C01840=1183.725,109.881,-51.815,-178.781,6.157,148.748
C01841=1183.720,110.129,-51.834,-178.778,6.158,148.748
C01842=1183.715,110.379,-51.854,-178.775,6.159,148.747
C01843=1183.710,110.628,-51.872,-178.773,6.160,148.747
C01844=1183.706,110.878,-51.891,-178.770,6.162,148.746
C01845=1183.701,111.126,-51.910,-178.767,6.163,148.746
C01846=1183.696,111.376,-51.929,-178.765,6.164,148.745
C01847=1183.691,111.625,-51.948,-178.762,6.166,148.745
C01848=1183.687,111.874,-51.967,-178.760,6.167,148.744
C01849=1183.682,112.123,-51.986,-178.757,6.168,148.744
C01850=1183.677,112.373,-52.005,-178.754,6.170,148.743
C01851=1183.672,112.622,-52.024,-178.752,6.171,148.743
C01852=1183.668,112.871,-52.043,-178.749,6.172,148.742
C01853=1183.662,113.120,-52.063,-178.746,6.174,148.742
C01854=1183.658,113.370,-52.081,-178.744,6.175,148.741
C01855=1183.653,113.619,-52.100,-178.741,6.177,148.741
C01856=1183.648,113.869,-52.120,-178.738,6.177,148.740
C01857=1183.643,114.117,-52.139,-178.736,6.179,148.740
C01858=1183.639,114.367,-52.158,-178.733,6.181,148.740
C01859=1183.634,114.616,-52.176,-178.730,6.181,148.739
C01860=1183.629,114.865,-52.196,-178.728,6.183,148.739
C01861=1183.624,115.114,-52.215,-178.726,6.184,148.738
C01862=1183.619,115.363,-52.234,-178.722,6.185,148.737
C01863=1183.614,115.612,-52.254,-178.720,6.187,148.737
C01864=1183.609,115.862,-52.273,-178.718,6.188,148.737
C01865=1183.605,116.110,-52.292,-178.714,6.189,148.736
C01866=1183.600,116.361,-52.311,-178.712,6.191,148.736
C01867=1183.594,116.610,-52.330,-178.710,6.192,148.735
C01868=1183.590,116.859,-52.349,-178.706,6.193,148.735
C01869=1183.585,117.108,-52.368,-178.704,6.195,148.734
C01870=1183.580,117.357,-52.388,-178.701,6.196,148.734
C01871=1183.576,117.607,-52.408,-178.698,6.197,148.733
C01872=1183.571,117.855,-52.427,-178.696,6.198,148.733
C01873=1183.566,118.105,-52.446,-178.693,6.200,148.732
C01874=1183.561,118.354,-52.465,-178.690,6.201,148.732
C01875=1183.556,118.603,-52.485,-178.688,6.202,148.731
C01876=1183.552,118.852,-52.504,-178.685,6.204,148.731
C01877=1183.547,119.101,-52.523,-178.683,6.206,148.731
C01878=1183.542,119.351,-52.543,-178.680,6.206,148.730
C01879=1183.537,119.600,-52.562,-178.677,6.208,148.729
C01880=1183.533,119.849,-52.581,-178.675,6.210,148.729
C01881=1183.527,120.098,-52.601,-178.672,6.210,148.728
C01882=1183.523,120.348,-52.620,-178.669,6.212,148.728
C01883=1183.518,120.597,-52.640,-178.667,6.214,148.728
C01884=1183.513,120.846,-52.659,-178.664,6.215,148.727
C01885=1183.509,121.095,-52.679,-178.661,6.216,148.727
C01886=1183.504,121.344,-52.699,-178.659,6.218,148.726
C01887=1183.499,121.593,-52.718,-178.657,6.219,148.726
C01888=1183.494,121.843,-52.738,-178.653,6.220,148.725
C01889=1183.489,122.092,-52.757,-178.651,6.222,148.725
C01890=1183.484,122.341,-52.777,-178.649,6.223,148.724
C01891=1183.480,122.590,-52.796,-178.645,6.224,148.724
C01892=1183.475,122.840,-52.815,-178.643,6.226,148.723
C01893=1183.470,123.088,-52.835,-178.641,6.227,148.723
C01894=1183.465,123.338,-52.855,-178.637,6.228,148.722
C01895=1183.461,123.587,-52.875,-178.635,6.230,148.722
C01896=1183.455,123.836,-52.894,-178.633,6.231,148.722
C01897=1183.451,124.086,-52.914,-178.630,6.233,148.721
C01898=1183.446,124.335,-52.934,-178.627,6.234,148.721
C01899=1183.441,124.584,-52.953,-178.624,6.236,148.720
C01900=1183.437,124.833,-52.972,-178.622,6.237,148.720
C01901=1183.432,125.082,-52.992,-178.619,6.239,148.719
C01902=1183.427,125.331,-53.012,-178.616,6.240,148.719
C01903=1183.422,125.580,-53.032,-178.614,6.241,148.718
C01904=1183.417,125.830,-53.051,-178.611,6.243,148.718
C01905=1183.413,126.079,-53.072,-178.608,6.244,148.717
C01906=1183.408,126.328,-53.091,-178.606,6.245,148.717
C01907=1183.403,126.577,-53.111,-178.603,6.247,148.716
C01908=1183.399,126.826,-53.131,-178.600,6.249,148.716
C01909=1183.394,127.076,-53.151,-178.597,6.250,148.715
C01910=1183.388,127.325,-53.170,-178.595,6.251,148.715
C01911=1183.384,127.574,-53.190,-178.592,6.253,148.715
C01912=1183.379,127.823,-53.210,-178.590,6.254,148.714
C01913=1183.375,128.073,-53.230,-178.587,6.255,148.714
C01914=1183.369,128.321,-53.250,-178.584,6.257,148.713
C01915=1183.365,128.570,-53.269,-178.582,6.258,148.713
C01916=1183.360,128.819,-53.290,-178.579,6.260,148.712
C01917=1183.356,129.069,-53.309,-178.576,6.261,148.712
C01918=1183.350,129.318,-53.329,-178.574,6.263,148.711
C01919=1183.346,129.567,-53.349,-178.571,6.264,148.711
C01920=1183.341,129.816,-53.369,-178.569,6.265,148.711
C01921=1183.337,130.065,-53.389,-178.566,6.267,148.710
C01922=1183.332,130.315,-53.409,-178.563,6.268,148.710
C01923=1183.327,130.563,-53.429,-178.560,6.270,148.709
C01924=1183.321,130.813,-53.449,-178.558,6.271,148.709
C01925=1183.317,131.062,-53.469,-178.555,6.272,148.708
C01926=1183.312,131.312,-53.489,-178.552,6.274,148.708
C01927=1183.308,131.560,-53.509,-178.550,6.276,148.707
C01928=1183.302,131.809,-53.529,-178.548,6.277,148.707
C01929=1183.298,132.058,-53.549,-178.544,6.278,148.706
C01930=1183.292,132.327,-53.571,-178.542,6.280,148.706
C01931=1183.288,132.595,-53.593,-178.539,6.282,148.706
C01932=1183.282,132.864,-53.614,-178.536,6.283,148.705
C01933=1183.277,133.133,-53.635,-178.533,6.285,148.705
C01934=1183.273,133.382,-53.656,-178.530,6.287,148.704
C01935=1183.268,133.631,-53.676,-178.528,6.287,148.704
C01936=1183.263,133.881,-53.696,-178.525,6.289,148.703
C01937=1183.258,134.130,-53.717,-178.522,6.291,148.703
C01938=1183.254,134.379,-53.736,-178.520,6.293,148.702
C01939=1183.249,134.628,-53.757,-178.517,6.293,148.702
C01940=1183.244,134.876,-53.777,-178.514,6.295,148.701
C01941=1183.239,135.126,-53.797,-178.512,6.297,148.701
C01942=1183.234,135.375,-53.817,-178.509,6.298,148.701
C01943=1183.230,135.624,-53.838,-178.507,6.299,148.700
C01944=1183.225,135.873,-53.858,-178.504,6.301,148.700
C01945=1183.220,136.123,-53.878,-178.501,6.302,148.699
C01946=1183.215,136.372,-53.899,-178.498,6.304,148.699
C01947=1183.211,136.621,-53.919,-178.496,6.306,148.698
C01948=1183.206,136.870,-53.939,-178.493,6.307,148.698
C01949=1183.201,137.120,-53.960,-178.490,6.308,148.697
C01950=1183.197,137.369,-53.980,-178.488,6.310,148.697
C01951=1183.192,137.617,-54.000,-178.485,6.312,148.697
C01952=1183.187,137.866,-54.020,-178.483,6.313,148.696
C01953=1183.182,138.116,-54.041,-178.480,6.315,148.696
C01954=1183.177,138.365,-54.061,-178.477,6.316,148.695
C01955=1183.173,138.614,-54.081,-178.474,6.318,148.695
C01956=1183.168,138.863,-54.102,-178.472,6.319,148.695
C01957=1183.163,139.112,-54.123,-178.469,6.320,148.694
C01958=1183.159,139.361,-54.143,-178.467,6.322,148.694
C01959=1183.153,139.611,-54.163,-178.464,6.324,148.693
C01960=1183.149,139.860,-54.184,-178.461,6.325,148.693
C01961=1183.144,140.109,-54.204,-178.459,6.326,148.692
C01962=1183.139,140.358,-54.225,-178.456,6.328,148.692
C01963=1183.135,140.607,-54.245,-178.453,6.330,148.692
C01964=1183.130,140.856,-54.266,-178.451,6.332,148.691
C01965=1183.125,141.105,-54.287,-178.447,6.333,148.691
C01966=1183.121,141.354,-54.307,-178.445,6.334,148.690
C01967=1183.116,141.603,-54.328,-178.443,6.336,148.690
C01968=1183.111,141.852,-54.349,-178.440,6.337,148.689
C01969=1183.107,142.101,-54.369,-178.437,6.339,148.689
C01970=1183.101,142.350,-54.390,-178.434,6.341,148.688
C01971=1183.097,142.599,-54.410,-178.431,6.342,148.688
C01972=1183.092,142.849,-54.431,-178.429,6.343,148.688
C01973=1183.087,143.098,-54.452,-178.427,6.345,148.687
C01974=1183.083,143.346,-54.472,-178.424,6.347,148.687
C01975=1183.078,143.596,-54.493,-178.421,6.349,148.686
C01976=1183.073,143.845,-54.513,-178.418,6.350,148.686
C01977=1183.068,144.094,-54.534,-178.416,6.351,148.685
C01978=1183.064,144.343,-54.555,-178.413,6.353,148.685
C01979=1183.059,144.592,-54.576,-178.411,6.354,148.685
C01980=1183.055,144.842,-54.596,-178.408,6.356,148.684
C01981=1183.050,145.091,-54.617,-178.405,6.358,148.684
C01982=1183.045,145.340,-54.638,-178.402,6.360,148.684
C01983=1183.040,145.589,-54.659,-178.400,6.360,148.683
C01984=1183.036,145.838,-54.679,-178.397,6.362,148.683
C01985=1183.031,146.087,-54.701,-178.395,6.364,148.682
C01986=1183.026,146.336,-54.721,-178.392,6.366,148.682
C01987=1183.021,146.585,-54.742,-178.389,6.367,148.681
C01988=1183.017,146.834,-54.762,-178.386,6.369,148.681
C01989=1183.011,147.083,-54.783,-178.384,6.370,148.681
C01990=1183.006,147.333,-54.804,-178.381,6.371,148.680
C01991=1183.003,147.582,-54.826,-178.378,6.373,148.680
C01992=1182.998,147.831,-54.847,-178.376,6.375,148.679
C01993=1182.993,148.080,-54.867,-178.373,6.377,148.679
C01994=1182.988,148.329,-54.888,-178.370,6.378,148.678
C01995=1182.984,148.577,-54.909,-178.368,6.380,148.678
C01996=1182.979,148.827,-54.930,-178.366,6.381,148.678
C01997=1182.973,149.076,-54.951,-178.362,6.383,148.677
C01998=1182.970,149.326,-54.972,-178.360,6.384,148.677
C01999=1182.965,149.574,-54.994,-178.357,6.386,148.676
C02000=1182.960,149.823,-55.014,-178.354,6.388,148.676
C02001=1182.955,150.072,-55.035,-178.352,6.390,148.676
C02002=1182.950,150.321,-55.057,-178.349,6.391,148.675
C02003=1182.945,150.570,-55.078,-178.347,6.392,148.675
C02004=1182.941,150.819,-55.098,-178.344,6.394,148.674
C02005=1182.936,151.069,-55.120,-178.342,6.396,148.674
C02006=1182.931,151.318,-55.141,-178.338,6.397,148.673
C02007=1182.927,151.567,-55.161,-178.336,6.399,148.673
C02008=1182.922,151.815,-55.183,-178.333,6.401,148.673
C02009=1182.917,152.065,-55.204,-178.330,6.403,148.672
C02010=1182.913,152.314,-55.225,-178.328,6.404,148.672
C02011=1182.908,152.563,-55.246,-178.325,6.405,148.672
C02012=1182.903,152.812,-55.267,-178.323,6.407,148.671
C02013=1182.898,153.061,-55.289,-178.320,6.409,148.671
C02014=1182.894,153.310,-55.309,-178.317,6.411,148.670
C02015=1182.889,153.559,-55.331,-178.314,6.412,148.670
C02016=1182.884,153.808,-55.352,-178.312,6.414,148.669
C02017=1182.879,154.057,-55.374,-178.309,6.416,148.669
C02018=1182.875,154.306,-55.394,-178.306,6.417,148.669
C02019=1182.871,154.555,-55.416,-178.304,6.418,148.668
C02020=1182.865,154.805,-55.437,-178.301,6.420,148.668
C02021=1182.861,155.053,-55.459,-178.299,6.422,148.668
C02022=1182.856,155.302,-55.480,-178.296,6.424,148.667
C02023=1182.852,155.552,-55.502,-178.293,6.425,148.667
C02024=1182.847,155.801,-55.523,-178.291,6.427,148.666
C02025=1182.842,156.049,-55.544,-178.288,6.429,148.666
C02026=1182.837,156.299,-55.565,-178.285,6.431,148.666
C02027=1182.832,156.548,-55.587,-178.282,6.432,148.665
C02028=1182.828,156.796,-55.608,-178.279,6.434,148.665
C02029=1182.823,157.046,-55.629,-178.277,6.436,148.664
C02030=1182.819,157.295,-55.651,-178.275,6.437,148.664
C02031=1182.814,157.544,-55.672,-178.272,6.438,148.664
C02032=1182.809,157.793,-55.694,-178.269,6.440,148.663
C02033=1182.804,158.041,-55.716,-178.267,6.442,148.663
C02034=1182.799,158.311,-55.738,-178.264,6.444,148.662
C02035=1182.794,158.580,-55.762,-178.261,6.445,148.662
C02036=1182.789,158.848,-55.785,-178.257,6.448,148.661
C02037=1182.784,159.118,-55.809,-178.255,6.449,148.661
C02038=1182.779,159.367,-55.831,-178.252,6.451,148.661
C02039=1182.774,159.616,-55.852,-178.249,6.453,148.660
C02040=1182.770,159.865,-55.873,-178.247,6.455,148.660
C02041=1182.766,160.114,-55.895,-178.244,6.456,148.660
C02042=1182.761,160.363,-55.916,-178.242,6.457,148.659
C02043=1182.756,160.612,-55.937,-178.239,6.459,148.659
C02044=1182.752,160.861,-55.959,-178.237,6.461,148.658
C02045=1182.747,161.110,-55.981,-178.234,6.463,148.658
C02046=1182.742,161.358,-56.003,-178.231,6.464,148.658
C02047=1182.738,161.608,-56.025,-178.229,6.466,148.657
C02048=1182.732,161.857,-56.046,-178.226,6.468,148.657
C02049=1182.728,162.106,-56.068,-178.223,6.470,148.657
C02050=1182.723,162.355,-56.090,-178.220,6.471,148.656
C02051=1182.718,162.604,-56.111,-178.217,6.473,148.656
C02052=1182.714,162.853,-56.133,-178.215,6.475,148.655
C02053=1182.709,163.102,-56.155,-178.212,6.477,148.655
C02054=1182.705,163.352,-56.176,-178.209,6.478,148.655
C02055=1182.700,163.600,-56.198,-178.207,6.480,148.654
C02056=1182.695,163.849,-56.220,-178.204,6.482,148.654
C02057=1182.691,164.098,-56.242,-178.201,6.484,148.653
C02058=1182.686,164.347,-56.263,-178.199,6.485,148.653
C02059=1182.681,164.596,-56.285,-178.196,6.487,148.653
C02060=1182.676,164.845,-56.308,-178.193,6.489,148.652
C02061=1182.672,165.095,-56.330,-178.191,6.490,148.652
C02062=1182.667,165.343,-56.351,-178.188,6.492,148.652
C02063=1182.662,165.592,-56.373,-178.186,6.493,148.651
C02064=1182.658,165.841,-56.395,-178.183,6.495,148.651
C02065=1182.653,166.090,-56.417,-178.180,6.497,148.650
C02066=1182.648,166.339,-56.439,-178.178,6.499,148.650
C02067=1182.644,166.588,-56.461,-178.175,6.501,148.650
C02068=1182.639,166.837,-56.483,-178.172,6.502,148.649
C02069=1182.634,167.086,-56.504,-178.170,6.504,148.649
C02070=1182.629,167.335,-56.527,-178.167,6.506,148.649
C02071=1182.625,167.584,-56.549,-178.164,6.508,148.648
C02072=1182.620,167.833,-56.571,-178.162,6.509,148.648
C02073=1182.615,168.082,-56.592,-178.159,6.511,148.648
C02074=1182.611,168.331,-56.615,-178.156,6.513,148.647
C02075=1182.606,168.580,-56.637,-178.154,6.515,148.647
C02076=1182.602,168.829,-56.659,-178.151,6.516,148.646
C02077=1182.597,169.078,-56.681,-178.148,6.518,148.646
C02078=1182.592,169.327,-56.703,-178.146,6.520,148.646
C02079=1182.588,169.576,-56.725,-178.143,6.522,148.645
C02080=1182.583,169.825,-56.748,-178.140,6.524,148.645
C02081=1182.578,170.073,-56.770,-178.137,6.525,148.645
C02082=1182.574,170.323,-56.792,-178.135,6.527,148.644
C02083=1182.569,170.571,-56.814,-178.132,6.529,148.644
C02084=1182.564,170.821,-56.836,-178.129,6.531,148.643
C02085=1182.559,171.070,-56.858,-178.127,6.532,148.643
C02086=1182.555,171.318,-56.881,-178.124,6.534,148.643
C02087=1182.551,171.568,-56.903,-178.121,6.536,148.642
C02088=1182.545,171.817,-56.925,-178.119,6.538,148.642
C02089=1182.541,172.066,-56.947,-178.116,6.540,148.642
C02090=1182.536,172.314,-56.970,-178.113,6.541,148.641
C02091=1182.531,172.564,-56.992,-178.111,6.543,148.641
C02092=1182.526,172.812,-57.014,-178.108,6.545,148.641
C02093=1182.523,173.061,-57.037,-178.105,6.547,148.640
C02094=1182.518,173.311,-57.059,-178.103,6.549,148.640
C02095=1182.513,173.559,-57.081,-178.100,6.551,148.640
C02096=1182.509,173.808,-57.104,-178.098,6.552,148.639
C02097=1182.503,174.057,-57.126,-178.095,6.554,148.639
C02098=1182.499,174.306,-57.148,-178.092,6.556,148.639
C02099=1182.495,174.555,-57.171,-178.090,6.558,148.638
C02100=1182.489,174.804,-57.193,-178.087,6.560,148.638
C02101=1182.485,175.053,-57.216,-178.084,6.562,148.638
C02102=1182.480,175.302,-57.238,-178.081,6.564,148.637
C02103=1182.475,175.551,-57.260,-178.078,6.566,148.637
C02104=1182.471,175.800,-57.283,-178.076,6.567,148.636
C02105=1182.466,176.049,-57.306,-178.073,6.569,148.636
C02106=1182.462,176.297,-57.328,-178.070,6.571,148.636
C02107=1182.457,176.547,-57.351,-178.068,6.573,148.635
C02108=1182.453,176.796,-57.373,-178.065,6.575,148.635
C02109=1182.448,177.044,-57.395,-178.062,6.576,148.635
C02110=1182.443,177.293,-57.418,-178.060,6.578,148.634
C02111=1182.439,177.543,-57.440,-178.057,6.580,148.634
C02112=1182.434,177.791,-57.463,-178.055,6.582,148.634
C02113=1182.429,178.040,-57.486,-178.052,6.584,148.633
C02114=1182.425,178.289,-57.509,-178.050,6.586,148.633
C02115=1182.420,178.538,-57.531,-178.047,6.587,148.633
C02116=1182.415,178.787,-57.554,-178.044,6.589,148.632
C02117=1182.411,179.036,-57.577,-178.042,6.591,148.632
C02118=1182.406,179.285,-57.599,-178.039,6.593,148.632
C02119=1182.402,179.534,-57.622,-178.036,6.594,148.631
C02120=1182.397,179.783,-57.644,-178.033,6.597,148.631
C02121=1182.393,180.032,-57.667,-178.030,6.599,148.631
C02122=1182.387,180.280,-57.690,-178.028,6.601,148.630
C02123=1182.383,180.530,-57.712,-178.025,6.602,148.630
C02124=1182.378,180.779,-57.736,-178.023,6.605,148.630
C02125=1182.374,181.027,-57.758,-178.020,6.606,148.629
C02126=1182.369,181.276,-57.781,-178.017,6.608,148.629
C02127=1182.364,181.525,-57.804,-178.015,6.610,148.629
C02128=1182.360,181.774,-57.827,-178.012,6.612,148.628
C02129=1182.355,182.024,-57.849,-178.009,6.613,148.628
C02130=1182.351,182.272,-57.872,-178.007,6.615,148.628
C02131=1182.346,182.521,-57.895,-178.004,6.617,148.627
C02132=1182.341,182.770,-57.918,-178.001,6.619,148.627
C02133=1182.337,183.019,-57.940,-177.998,6.621,148.627
C02134=1182.332,183.267,-57.963,-177.996,6.624,148.626
C02135=1182.328,183.516,-57.986,-177.993,6.625,148.626
C02136=1182.323,183.765,-58.010,-177.991,6.627,148.626
C02137=1182.318,184.014,-58.033,-177.988,6.629,148.625
C02138=1182.314,184.284,-58.057,-177.985,6.631,148.625
C02139=1182.308,184.553,-58.082,-177.982,6.633,148.625
C02140=1182.303,184.823,-58.107,-177.979,6.635,148.624
C02141=1182.299,185.093,-58.132,-177.977,6.637,148.624
C02142=1182.294,185.342,-58.155,-177.974,6.639,148.624
C02143=1182.289,185.591,-58.179,-177.971,6.641,148.623
C02144=1182.285,185.839,-58.201,-177.968,6.643,148.623
C02145=1182.280,186.088,-58.224,-177.965,6.645,148.623
C02146=1182.275,186.337,-58.247,-177.963,6.647,148.622
C02147=1182.270,186.586,-58.270,-177.960,6.648,148.622
C02148=1182.266,186.835,-58.293,-177.958,6.650,148.622
C02149=1182.261,187.084,-58.317,-177.955,6.652,148.621
C02150=1182.257,187.333,-58.340,-177.952,6.654,148.621
C02151=1182.251,187.582,-58.363,-177.949,6.657,148.621
C02152=1182.248,187.830,-58.386,-177.947,6.658,148.620
C02153=1182.243,188.079,-58.409,-177.944,6.660,148.620
C02154=1182.238,188.328,-58.432,-177.941,6.662,148.620
C02155=1182.233,188.577,-58.456,-177.939,6.664,148.619
C02156=1182.229,188.826,-58.478,-177.936,6.666,148.619
C02157=1182.225,189.075,-58.502,-177.934,6.668,148.619
C02158=1182.220,189.324,-58.525,-177.931,6.670,148.618
C02159=1182.215,189.573,-58.548,-177.928,6.672,148.618
C02160=1182.210,189.822,-58.572,-177.925,6.674,148.618
C02161=1182.206,190.070,-58.596,-177.923,6.676,148.618
C02162=1182.202,190.319,-58.618,-177.920,6.678,148.617
C02163=1182.197,190.568,-58.642,-177.918,6.680,148.617
C02164=1182.192,190.817,-58.665,-177.915,6.681,148.617
C02165=1182.188,191.066,-58.688,-177.912,6.683,148.616
C02166=1182.183,191.315,-58.712,-177.909,6.686,148.616
C02167=1182.178,191.564,-58.735,-177.907,6.688,148.616
C02168=1182.174,191.813,-58.759,-177.904,6.690,148.615
C02169=1182.169,192.061,-58.783,-177.901,6.692,148.615
C02170=1182.164,192.310,-58.806,-177.899,6.693,148.615
C02171=1182.160,192.559,-58.829,-177.896,6.695,148.614
C02172=1182.156,192.808,-58.852,-177.893,6.697,148.614
C02173=1182.151,193.057,-58.875,-177.891,6.700,148.614
C02174=1182.147,193.306,-58.900,-177.888,6.702,148.613
C02175=1182.142,193.555,-58.923,-177.885,6.703,148.613
C02176=1182.137,193.804,-58.946,-177.883,6.705,148.613
C02177=1182.133,194.053,-58.970,-177.880,6.707,148.612
C02178=1182.128,194.301,-58.994,-177.878,6.709,148.612
C02179=1182.123,194.550,-59.017,-177.875,6.712,148.612
C02180=1182.119,194.799,-59.040,-177.872,6.714,148.612
C02181=1182.114,195.048,-59.064,-177.869,6.715,148.611
C02182=1182.110,195.297,-59.088,-177.867,6.717,148.611
C02183=1182.105,195.546,-59.111,-177.864,6.719,148.611
C02184=1182.101,195.794,-59.135,-177.861,6.722,148.610
C02185=1182.096,196.043,-59.159,-177.859,6.724,148.610
C02186=1182.091,196.292,-59.182,-177.856,6.725,148.610
C02187=1182.087,196.540,-59.206,-177.853,6.727,148.609
C02188=1182.082,196.790,-59.229,-177.851,6.729,148.609
C02189=1182.078,197.038,-59.253,-177.848,6.731,148.609
C02190=1182.073,197.287,-59.277,-177.845,6.734,148.609
C02191=1182.068,197.536,-59.300,-177.842,6.736,148.608
C02192=1182.064,197.784,-59.324,-177.840,6.737,148.608
C02193=1182.058,198.034,-59.348,-177.838,6.739,148.608
C02194=1182.054,198.282,-59.372,-177.835,6.741,148.607
C02195=1182.049,198.531,-59.396,-177.832,6.744,148.607
C02196=1182.045,198.780,-59.420,-177.829,6.746,148.607
C02197=1182.040,199.029,-59.443,-177.827,6.748,148.607
C02198=1182.036,199.278,-59.468,-177.824,6.750,148.606
C02199=1182.032,199.527,-59.491,-177.822,6.751,148.606
C02200=1182.027,199.775,-59.515,-177.818,6.754,148.606
C02201=1182.022,200.025,-59.539,-177.816,6.756,148.605
C02202=1182.018,200.273,-59.563,-177.813,6.758,148.605
C02203=1182.013,200.522,-59.586,-177.811,6.760,148.605
C02204=1182.008,200.770,-59.610,-177.808,6.762,148.604
C02205=1182.004,201.019,-59.635,-177.805,6.764,148.604
C02206=1181.999,201.268,-59.658,-177.803,6.766,148.604
C02207=1181.995,201.517,-59.683,-177.800,6.768,148.604
C02208=1181.990,201.766,-59.706,-177.797,6.770,148.603
C02209=1181.986,202.015,-59.730,-177.794,6.772,148.603
C02210=1181.981,202.263,-59.754,-177.792,6.775,148.603
C02211=1181.977,202.512,-59.778,-177.789,6.776,148.603
C02212=1181.972,202.761,-59.802,-177.787,6.778,148.602
C02213=1181.968,203.010,-59.827,-177.784,6.780,148.602
C02214=1181.963,203.259,-59.850,-177.781,6.783,148.602
C02215=1181.959,203.507,-59.874,-177.779,6.785,148.601
C02216=1181.953,203.756,-59.899,-177.776,6.787,148.601
C02217=1181.949,204.005,-59.923,-177.773,6.788,148.601
C02218=1181.944,204.254,-59.946,-177.770,6.791,148.601
C02219=1181.941,204.503,-59.971,-177.768,6.793,148.600
C02220=1181.935,204.751,-59.996,-177.765,6.795,148.600
C02221=1181.931,205.000,-60.020,-177.762,6.797,148.600
C02222=1181.926,205.249,-60.043,-177.760,6.800,148.600
C02223=1181.922,205.498,-60.068,-177.757,6.801,148.599
C02224=1181.917,205.747,-60.092,-177.754,6.803,148.599
C02225=1181.913,205.995,-60.116,-177.752,6.805,148.599
C02226=1181.908,206.244,-60.141,-177.749,6.808,148.598
C02227=1181.904,206.492,-60.165,-177.746,6.810,148.598
C02228=1181.899,206.742,-60.189,-177.744,6.812,148.598
C02229=1181.894,206.991,-60.213,-177.741,6.814,148.598
C02230=1181.890,207.239,-60.237,-177.738,6.816,148.597
C02231=1181.886,207.488,-60.261,-177.736,6.818,148.597
C02232=1181.881,207.737,-60.286,-177.733,6.820,148.597
C02233=1181.877,207.985,-60.311,-177.731,6.822,148.596
C02234=1181.871,208.234,-60.335,-177.727,6.825,148.596
C02235=1181.867,208.483,-60.359,-177.725,6.827,148.596
C02236=1181.863,208.732,-60.384,-177.723,6.829,148.596
C02237=1181.858,208.980,-60.408,-177.720,6.830,148.595
C02238=1181.854,209.229,-60.432,-177.717,6.833,148.595
C02239=1181.849,209.478,-60.458,-177.715,6.835,148.595
C02240=1181.845,209.727,-60.482,-177.712,6.837,148.595
C02241=1181.840,209.975,-60.506,-177.709,6.840,148.594
C02242=1181.834,210.246,-60.532,-177.706,6.841,148.594
C02243=1181.830,210.517,-60.559,-177.703,6.844,148.594
C02244=1181.825,210.787,-60.585,-177.701,6.846,148.594
C02245=1181.820,211.057,-60.612,-177.697,6.849,148.593
C02246=1181.816,211.306,-60.637,-177.695,6.851,148.593
C02247=1181.811,211.555,-60.661,-177.693,6.853,148.593
C02248=1181.806,211.804,-60.686,-177.689,6.855,148.592
C02249=1181.802,212.053,-60.710,-177.687,6.857,148.592
C02250=1181.797,212.301,-60.735,-177.684,6.859,148.592
C02251=1181.793,212.549,-60.760,-177.681,6.862,148.592
C02252=1181.789,212.799,-60.785,-177.679,6.864,148.591
C02253=1181.783,213.047,-60.810,-177.676,6.866,148.591
C02254=1181.779,213.296,-60.834,-177.674,6.868,148.591
C02255=1181.774,213.545,-60.859,-177.670,6.870,148.591
C02256=1181.770,213.794,-60.883,-177.668,6.872,148.590
C02257=1181.766,214.042,-60.908,-177.666,6.874,148.590
C02258=1181.761,214.291,-60.933,-177.662,6.877,148.590
C02259=1181.756,214.540,-60.957,-177.660,6.879,148.590
C02260=1181.752,214.789,-60.982,-177.658,6.881,148.589
C02261=1181.748,215.037,-61.007,-177.654,6.883,148.589
C02262=1181.743,215.286,-61.032,-177.652,6.886,148.589
C02263=1181.739,215.535,-61.056,-177.650,6.887,148.589
C02264=1181.734,215.783,-61.081,-177.646,6.890,148.588
C02265=1181.729,216.032,-61.107,-177.644,6.892,148.588
C02266=1181.725,216.281,-61.131,-177.641,6.894,148.588
C02267=1181.720,216.530,-61.156,-177.638,6.897,148.588
C02268=1181.716,216.778,-61.181,-177.636,6.899,148.587
C02269=1181.712,217.027,-61.206,-177.633,6.901,148.587
C02270=1181.707,217.276,-61.230,-177.631,6.903,148.587
C02271=1181.702,217.524,-61.256,-177.628,6.905,148.587
C02272=1181.698,217.773,-61.280,-177.625,6.907,148.586
C02273=1181.693,218.021,-61.305,-177.623,6.910,148.586
C02274=1181.689,218.271,-61.330,-177.620,6.912,148.586
C02275=1181.684,218.519,-61.355,-177.617,6.914,148.586
C02276=1181.680,218.768,-61.380,-177.615,6.917,148.585
C02277=1181.675,219.017,-61.405,-177.612,6.918,148.585
C02278=1181.671,219.265,-61.431,-177.610,6.921,148.585
C02279=1181.666,219.514,-61.455,-177.606,6.923,148.585
C02280=1181.662,219.763,-61.480,-177.604,6.925,148.584
C02281=1181.657,220.011,-61.505,-177.602,6.927,148.584
C02282=1181.653,220.260,-61.531,-177.598,6.930,148.584
C02283=1181.648,220.509,-61.556,-177.596,6.932,148.584
C02284=1181.644,220.757,-61.581,-177.594,6.934,148.584
C02285=1181.639,221.006,-61.605,-177.590,6.936,148.583
C02286=1181.635,221.255,-61.631,-177.588,6.938,148.583
C02287=1181.630,221.504,-61.656,-177.586,6.940,148.583
C02288=1181.625,221.752,-61.682,-177.583,6.943,148.583
C02289=1181.620,222.001,-61.706,-177.580,6.945,148.582
C02290=1181.617,222.250,-61.731,-177.577,6.947,148.582
C02291=1181.613,222.498,-61.757,-177.575,6.950,148.582
C02292=1181.608,222.747,-61.782,-177.572,6.952,148.582
C02293=1181.603,222.996,-61.808,-177.570,6.954,148.582
C02294=1181.598,223.244,-61.833,-177.567,6.956,148.581
C02295=1181.594,223.494,-61.858,-177.564,6.958,148.581
C02296=1181.589,223.742,-61.883,-177.561,6.961,148.581
C02297=1181.585,223.990,-61.909,-177.559,6.963,148.580
C02298=1181.581,224.240,-61.934,-177.556,6.965,148.580
C02299=1181.576,224.488,-61.959,-177.553,6.968,148.580
C02300=1181.572,224.736,-61.985,-177.551,6.970,148.580
C02301=1181.567,224.985,-62.009,-177.548,6.972,148.580
C02302=1181.563,225.234,-62.035,-177.545,6.974,148.579
C02303=1181.558,225.482,-62.061,-177.543,6.976,148.579
C02304=1181.554,225.731,-62.086,-177.540,6.979,148.579
C02305=1181.549,225.980,-62.111,-177.538,6.981,148.579
C02306=1181.544,226.228,-62.137,-177.535,6.983,148.578
C02307=1181.540,226.477,-62.162,-177.532,6.986,148.578
C02308=1181.536,226.726,-62.188,-177.530,6.988,148.578
C02309=1181.531,226.974,-62.214,-177.527,6.991,148.578
C02310=1181.526,227.224,-62.239,-177.524,6.993,148.578
C02311=1181.522,227.472,-62.264,-177.522,6.995,148.578
C02312=1181.517,227.720,-62.290,-177.519,6.997,148.577
C02313=1181.513,227.969,-62.315,-177.516,6.999,148.577
C02314=1181.508,228.217,-62.341,-177.513,7.002,148.577
C02315=1181.504,228.466,-62.367,-177.511,7.004,148.577
C02316=1181.500,228.715,-62.392,-177.508,7.006,148.576
C02317=1181.496,228.964,-62.418,-177.505,7.009,148.576
C02318=1181.491,229.212,-62.444,-177.503,7.011,148.576
C02319=1181.487,229.461,-62.469,-177.500,7.014,148.576
C02320=1181.482,229.710,-62.494,-177.498,7.016,148.576
C02321=1181.477,229.959,-62.520,-177.495,7.017,148.575
C02322=1181.472,230.207,-62.546,-177.492,7.020,148.575
C02323=1181.468,230.456,-62.572,-177.490,7.022,148.575
C02324=1181.463,230.704,-62.597,-177.487,7.025,148.575
C02325=1181.459,230.953,-62.623,-177.484,7.027,148.574
C02326=1181.455,231.202,-62.649,-177.482,7.029,148.574
C02327=1181.451,231.450,-62.675,-177.479,7.032,148.574
C02328=1181.446,231.698,-62.701,-177.477,7.034,148.574
C02329=1181.441,231.947,-62.727,-177.473,7.037,148.574
C02330=1181.437,232.196,-62.753,-177.471,7.039,148.574
C02331=1181.432,232.444,-62.778,-177.468,7.041,148.573
C02332=1181.428,232.693,-62.804,-177.466,7.044,148.573
C02333=1181.424,232.942,-62.829,-177.463,7.045,148.573
C02334=1181.419,233.191,-62.855,-177.460,7.048,148.573
C02335=1181.414,233.440,-62.882,-177.458,7.050,148.572
C02336=1181.410,233.688,-62.907,-177.455,7.053,148.572
C02337=1181.406,233.936,-62.933,-177.452,7.055,148.572
C02338=1181.401,234.185,-62.959,-177.450,7.058,148.572
C02339=1181.396,234.434,-62.986,-177.447,7.060,148.572
C02340=1181.392,234.682,-63.011,-177.444,7.063,148.572
C02341=1181.387,234.931,-63.037,-177.442,7.065,148.571
C02342=1181.384,235.179,-63.063,-177.439,7.067,148.571
C02343=1181.379,235.428,-63.089,-177.437,7.070,148.571
C02344=1181.374,235.677,-63.115,-177.434,7.071,148.571
C02345=1181.370,235.925,-63.141,-177.431,7.074,148.571
C02346=1181.365,236.196,-63.169,-177.428,7.077,148.570
C02347=1181.360,236.469,-63.198,-177.426,7.079,148.570
C02348=1181.355,236.740,-63.227,-177.423,7.082,148.570
C02349=1181.351,237.012,-63.255,-177.420,7.084,148.570
C02350=1181.346,237.260,-63.282,-177.417,7.087,148.570
C02351=1181.341,237.508,-63.307,-177.415,7.090,148.570
C02352=1181.337,237.757,-63.333,-177.412,7.091,148.569
C02353=1181.332,238.006,-63.360,-177.409,7.094,148.569
C02354=1181.328,238.254,-63.386,-177.407,7.096,148.569
C02355=1181.324,238.503,-63.412,-177.404,7.099,148.569
C02356=1181.319,238.752,-63.439,-177.401,7.101,148.568
C02357=1181.315,239.001,-63.464,-177.398,7.104,148.568
C02358=1181.310,239.248,-63.491,-177.396,7.106,148.568
C02359=1181.305,239.497,-63.517,-177.393,7.109,148.568
C02360=1181.301,239.746,-63.543,-177.391,7.111,148.568
C02361=1181.297,239.994,-63.570,-177.388,7.113,148.568
C02362=1181.292,240.243,-63.595,-177.386,7.116,148.567
C02363=1181.288,240.492,-63.622,-177.382,7.118,148.567
C02364=1181.283,240.741,-63.648,-177.380,7.120,148.567
C02365=1181.280,240.989,-63.675,-177.377,7.123,148.567
C02366=1181.275,241.238,-63.701,-177.375,7.125,148.567
C02367=1181.271,241.486,-63.727,-177.372,7.128,148.567
C02368=1181.265,241.734,-63.753,-177.370,7.130,148.567
C02369=1181.261,241.983,-63.780,-177.367,7.133,148.566
C02370=1181.257,242.231,-63.807,-177.364,7.135,148.566
C02371=1181.252,242.480,-63.833,-177.361,7.138,148.566
C02372=1181.248,242.728,-63.860,-177.359,7.140,148.566
C02373=1181.243,242.977,-63.886,-177.356,7.143,148.566
C02374=1181.239,243.226,-63.913,-177.354,7.145,148.565
C02375=1181.235,243.474,-63.939,-177.351,7.148,148.565
C02376=1181.230,243.723,-63.965,-177.348,7.149,148.565
C02377=1181.226,243.971,-63.992,-177.346,7.152,148.565
C02378=1181.221,244.220,-64.019,-177.343,7.155,148.565
C02379=1181.216,244.469,-64.045,-177.340,7.157,148.565
C02380=1181.212,244.717,-64.072,-177.338,7.159,148.564
C02381=1181.208,244.965,-64.099,-177.335,7.162,148.564
C02382=1181.204,245.214,-64.125,-177.333,7.164,148.564
C02383=1181.199,245.463,-64.152,-177.330,7.167,148.564
C02384=1181.195,245.711,-64.178,-177.328,7.169,148.564
C02385=1181.190,245.959,-64.205,-177.324,7.172,148.564
C02386=1181.185,246.209,-64.232,-177.322,7.174,148.564
C02387=1181.181,246.457,-64.258,-177.320,7.177,148.563
C02388=1181.177,246.705,-64.285,-177.317,7.179,148.563
C02389=1181.172,246.954,-64.312,-177.314,7.182,148.563
C02390=1181.168,247.202,-64.339,-177.312,7.184,148.563
C02391=1181.163,247.451,-64.365,-177.309,7.187,148.563
C02392=1181.159,247.700,-64.392,-177.307,7.189,148.563
C02393=1181.155,247.948,-64.418,-177.304,7.192,148.563
C02394=1181.150,248.196,-64.446,-177.301,7.194,148.562
C02395=1181.145,248.445,-64.473,-177.298,7.197,148.562
C02396=1181.142,248.694,-64.499,-177.296,7.200,148.562
C02397=1181.137,248.942,-64.526,-177.293,7.201,148.562
C02398=1181.133,249.191,-64.554,-177.290,7.204,148.562
C02399=1181.128,249.439,-64.579,-177.288,7.206,148.562
C02400=1181.124,249.688,-64.606,-177.285,7.209,148.561
C02401=1181.119,249.936,-64.633,-177.283,7.211,148.561
C02402=1181.115,250.185,-64.660,-177.280,7.214,148.561
C02403=1181.111,250.433,-64.687,-177.278,7.216,148.561
C02404=1181.106,250.682,-64.714,-177.275,7.219,148.561
C02405=1181.101,250.930,-64.741,-177.272,7.222,148.561
C02406=1181.097,251.179,-64.768,-177.270,7.224,148.561
C02407=1181.093,251.428,-64.796,-177.267,7.227,148.560
C02408=1181.089,251.676,-64.822,-177.264,7.229,148.560
C02409=1181.084,251.924,-64.849,-177.262,7.232,148.560
C02410=1181.079,252.173,-64.876,-177.260,7.234,148.560
C02411=1181.075,252.421,-64.904,-177.256,7.237,148.560
C02412=1181.070,252.669,-64.931,-177.254,7.240,148.560
C02413=1181.066,252.917,-64.957,-177.251,7.242,148.560
C02414=1181.062,253.167,-64.985,-177.248,7.245,148.559
C02415=1181.058,253.415,-65.012,-177.246,7.247,148.559
C02416=1181.053,253.664,-65.039,-177.243,7.250,148.559
C02417=1181.048,253.912,-65.066,-177.241,7.252,148.559
C02418=1181.044,254.161,-65.093,-177.238,7.254,148.559
C02419=1181.039,254.409,-65.121,-177.235,7.257,148.559
C02420=1181.036,254.657,-65.148,-177.233,7.260,148.559
C02421=1181.031,254.906,-65.175,-177.230,7.263,148.559
C02422=1181.027,255.154,-65.202,-177.228,7.264,148.558
C02423=1181.022,255.403,-65.229,-177.225,7.267,148.558
C02424=1181.018,255.651,-65.257,-177.222,7.270,148.558
C02425=1181.014,255.900,-65.284,-177.220,7.272,148.558
C02426=1181.009,256.148,-65.311,-177.217,7.275,148.558
C02427=1181.004,256.397,-65.338,-177.215,7.277,148.558
C02428=1181.000,256.645,-65.366,-177.212,7.280,148.558
C02429=1180.996,256.894,-65.393,-177.209,7.283,148.558
C02430=1180.991,257.143,-65.420,-177.206,7.285,148.557
C02431=1180.987,257.390,-65.448,-177.204,7.288,148.557
C02432=1180.982,257.639,-65.475,-177.202,7.290,148.557
C02433=1180.978,257.888,-65.503,-177.199,7.293,148.557
C02434=1180.974,258.136,-65.531,-177.196,7.296,148.557
C02435=1180.969,258.384,-65.558,-177.193,7.298,148.557
C02436=1180.965,258.633,-65.585,-177.191,7.301,148.557
C02437=1180.961,258.882,-65.613,-177.189,7.303,148.557
C02438=1180.956,259.130,-65.640,-177.186,7.306,148.557
C02439=1180.952,259.378,-65.668,-177.183,7.309,148.557
C02440=1180.947,259.626,-65.695,-177.180,7.311,148.556
C02441=1180.943,259.875,-65.723,-177.178,7.314,148.556
C02442=1180.939,260.123,-65.750,-177.175,7.317,148.556
C02443=1180.934,260.371,-65.778,-177.173,7.319,148.556
C02444=1180.930,260.621,-65.805,-177.170,7.322,148.556
C02445=1180.926,260.869,-65.832,-177.167,7.324,148.556
C02446=1180.921,261.117,-65.861,-177.165,7.327,148.556
C02447=1180.917,261.366,-65.889,-177.162,7.330,148.556
C02448=1180.912,261.614,-65.916,-177.160,7.332,148.556
C02449=1180.908,261.862,-65.944,-177.157,7.335,148.556
C02450=1180.903,262.136,-65.974,-177.154,7.338,148.555
C02451=1180.898,262.408,-66.005,-177.151,7.341,148.555
C02452=1180.894,262.681,-66.035,-177.148,7.344,148.555
C02453=1180.889,262.954,-66.065,-177.145,7.346,148.555
C02454=1180.885,263.203,-66.092,-177.142,7.349,148.555
C02455=1180.880,263.451,-66.121,-177.140,7.351,148.555
C02456=1180.876,263.700,-66.149,-177.138,7.354,148.555
C02457=1180.871,263.948,-66.176,-177.135,7.357,148.555
C02458=1180.867,264.196,-66.204,-177.133,7.359,148.555
C02459=1180.863,264.445,-66.232,-177.130,7.362,148.555
C02460=1180.858,264.693,-66.259,-177.127,7.365,148.554
C02461=1180.854,264.942,-66.288,-177.125,7.367,148.554
C02462=1180.850,265.190,-66.315,-177.122,7.370,148.554
C02463=1180.845,265.438,-66.342,-177.119,7.373,148.554
C02464=1180.840,265.687,-66.371,-177.117,7.375,148.554
C02465=1180.836,265.935,-66.399,-177.114,7.378,148.554
C02466=1180.832,266.184,-66.427,-177.111,7.381,148.554
C02467=1180.827,266.433,-66.455,-177.109,7.383,148.554
C02468=1180.823,266.680,-66.483,-177.106,7.386,148.554
C02469=1180.819,266.929,-66.511,-177.103,7.389,148.553
C02470=1180.814,267.177,-66.538,-177.101,7.391,148.553
C02471=1180.810,267.426,-66.567,-177.098,7.394,148.553
C02472=1180.806,267.674,-66.595,-177.096,7.397,148.553
C02473=1180.802,267.923,-66.622,-177.094,7.399,148.553
C02474=1180.796,268.171,-66.651,-177.091,7.402,148.553
C02475=1180.793,268.420,-66.679,-177.088,7.405,148.553
C02476=1180.788,268.668,-66.707,-177.085,7.407,148.553
C02477=1180.783,268.916,-66.735,-177.083,7.410,148.553
C02478=1180.780,269.164,-66.763,-177.080,7.413,148.553
C02479=1180.774,269.412,-66.792,-177.078,7.415,148.553
C02480=1180.771,269.661,-66.820,-177.075,7.418,148.553
C02481=1180.766,269.909,-66.848,-177.072,7.421,148.553
C02482=1180.762,270.158,-66.876,-177.070,7.423,148.552
C02483=1180.758,270.406,-66.904,-177.067,7.426,148.552
C02484=1180.753,270.655,-66.933,-177.065,7.429,148.552
C02485=1180.749,270.902,-66.961,-177.062,7.432,148.552
C02486=1180.745,271.151,-66.989,-177.059,7.434,148.552
C02487=1180.740,271.400,-67.017,-177.057,7.437,148.552
C02488=1180.736,271.648,-67.045,-177.054,7.440,148.552
C02489=1180.732,271.897,-67.074,-177.052,7.442,148.552
C02490=1180.727,272.145,-67.102,-177.049,7.445,148.552
C02491=1180.723,272.393,-67.130,-177.046,7.448,148.552
C02492=1180.718,272.641,-67.158,-177.044,7.450,148.552
C02493=1180.714,272.890,-67.187,-177.041,7.453,148.552
C02494=1180.710,273.138,-67.215,-177.039,7.456,148.552
C02495=1180.705,273.387,-67.243,-177.036,7.459,148.552
C02496=1180.701,273.634,-67.272,-177.034,7.461,148.551
C02497=1180.697,273.883,-67.301,-177.031,7.464,148.551
C02498=1180.693,274.132,-67.329,-177.028,7.467,148.551
C02499=1180.688,274.380,-67.357,-177.026,7.469,148.551
C02500=1180.684,274.628,-67.385,-177.023,7.472,148.551
C02501=1180.679,274.876,-67.414,-177.020,7.475,148.551
C02502=1180.675,275.125,-67.443,-177.017,7.478,148.551
C02503=1180.671,275.373,-67.471,-177.015,7.480,148.551
C02504=1180.666,275.622,-67.500,-177.013,7.483,148.551
C02505=1180.662,275.870,-67.528,-177.010,7.486,148.551
C02506=1180.657,276.118,-67.557,-177.007,7.489,148.551
C02507=1180.653,276.367,-67.586,-177.005,7.492,148.551
C02508=1180.649,276.615,-67.614,-177.002,7.494,148.551
C02509=1180.644,276.863,-67.643,-176.999,7.497,148.551
C02510=1180.641,277.111,-67.671,-176.997,7.500,148.551
C02511=1180.636,277.360,-67.700,-176.995,7.503,148.550
C02512=1180.631,277.608,-67.729,-176.992,7.506,148.550
C02513=1180.628,277.856,-67.757,-176.989,7.509,148.550
C02514=1180.623,278.105,-67.786,-176.987,7.511,148.550
C02515=1180.618,278.353,-67.815,-176.984,7.514,148.550
C02516=1180.615,278.601,-67.843,-176.981,7.517,148.550
C02517=1180.610,278.850,-67.872,-176.979,7.520,148.550
C02518=1180.605,279.098,-67.901,-176.977,7.522,148.550
C02519=1180.602,279.346,-67.930,-176.974,7.525,148.550
C02520=1180.597,279.595,-67.958,-176.971,7.528,148.550
C02521=1180.592,279.843,-67.987,-176.968,7.531,148.550
C02522=1180.588,280.091,-68.016,-176.966,7.533,148.550
C02523=1180.584,280.340,-68.044,-176.964,7.536,148.550
C02524=1180.580,280.588,-68.074,-176.961,7.539,148.550
C02525=1180.575,280.836,-68.103,-176.958,7.542,148.550
C02526=1180.571,281.085,-68.132,-176.956,7.544,148.550
C02527=1180.567,281.332,-68.161,-176.953,7.547,148.550
C02528=1180.563,281.581,-68.189,-176.950,7.550,148.550
C02529=1180.558,281.829,-68.218,-176.948,7.553,148.550
C02530=1180.554,282.078,-68.247,-176.945,7.556,148.550
C02531=1180.549,282.326,-68.277,-176.943,7.558,148.549
C02532=1180.545,282.573,-68.305,-176.940,7.561,148.549
C02533=1180.541,282.822,-68.334,-176.937,7.564,148.549
C02534=1180.537,283.070,-68.363,-176.935,7.567,148.549
C02535=1180.532,283.319,-68.392,-176.932,7.569,148.549
C02536=1180.528,283.568,-68.421,-176.930,7.572,148.549
C02537=1180.523,283.815,-68.450,-176.927,7.575,148.549
C02538=1180.519,284.064,-68.479,-176.924,7.578,148.549
C02539=1180.515,284.312,-68.508,-176.922,7.580,148.549
C02540=1180.511,284.560,-68.538,-176.919,7.583,148.549
C02541=1180.506,284.808,-68.567,-176.917,7.586,148.549
C02542=1180.502,285.057,-68.595,-176.914,7.589,148.549
C02543=1180.498,285.305,-68.625,-176.912,7.593,148.549
C02544=1180.494,285.553,-68.654,-176.910,7.595,148.549
C02545=1180.489,285.802,-68.684,-176.907,7.598,148.549
C02546=1180.484,286.050,-68.712,-176.904,7.601,148.549
C02547=1180.480,286.298,-68.742,-176.901,7.604,148.549
C02548=1180.476,286.546,-68.771,-176.899,7.607,148.549
C02549=1180.472,286.795,-68.800,-176.896,7.609,148.549
C02550=1180.468,287.043,-68.830,-176.894,7.612,148.549
C02551=1180.463,287.291,-68.859,-176.891,7.615,148.549
C02552=1180.459,287.540,-68.888,-176.888,7.618,148.549
C02553=1180.454,287.788,-68.917,-176.886,7.621,148.549
C02554=1180.450,288.062,-68.950,-176.883,7.624,148.549
C02555=1180.445,288.337,-68.983,-176.880,7.627,148.549
C02556=1180.441,288.611,-69.015,-176.877,7.630,148.549
C02557=1180.436,288.887,-69.047,-176.875,7.633,148.549
C02558=1180.432,289.135,-69.077,-176.872,7.636,148.549
C02559=1180.427,289.382,-69.106,-176.869,7.639,148.549
C02560=1180.423,289.631,-69.135,-176.866,7.642,148.549
C02561=1180.419,289.879,-69.165,-176.864,7.645,148.549
C02562=1180.414,290.127,-69.194,-176.862,7.647,148.549
C02563=1180.410,290.375,-69.224,-176.859,7.650,148.549
C02564=1180.406,290.624,-69.253,-176.857,7.653,148.549
C02565=1180.402,290.872,-69.283,-176.854,7.656,148.549
C02566=1180.397,291.121,-69.313,-176.851,7.659,148.549
C02567=1180.393,291.369,-69.342,-176.848,7.662,148.549
C02568=1180.389,291.617,-69.372,-176.846,7.664,148.548
C02569=1180.384,291.865,-69.401,-176.843,7.667,148.548
C02570=1180.380,292.114,-69.431,-176.841,7.671,148.549
C02571=1180.376,292.362,-69.460,-176.838,7.674,148.549
C02572=1180.372,292.610,-69.490,-176.836,7.677,148.549
C02573=1180.367,292.857,-69.519,-176.834,7.679,148.548
C02574=1180.362,293.106,-69.549,-176.831,7.682,148.548
C02575=1180.358,293.354,-69.579,-176.828,7.685,148.548
C02576=1180.354,293.602,-69.608,-176.825,7.688,148.548
C02577=1180.350,293.850,-69.638,-176.823,7.691,148.548
C02578=1180.346,294.098,-69.668,-176.820,7.694,148.549
C02579=1180.341,294.347,-69.698,-176.818,7.696,148.548
C02580=1180.337,294.595,-69.727,-176.816,7.699,148.548
C02581=1180.333,294.843,-69.757,-176.813,7.702,148.548
C02582=1180.329,295.091,-69.787,-176.810,7.705,148.548
C02583=1180.324,295.339,-69.817,-176.807,7.708,148.548
C02584=1180.320,295.588,-69.847,-176.805,7.712,148.549
C02585=1180.316,295.835,-69.877,-176.803,7.714,148.548
C02586=1180.312,296.084,-69.907,-176.800,7.717,148.548
C02587=1180.307,296.333,-69.937,-176.798,7.720,148.548
C02588=1180.303,296.581,-69.967,-176.795,7.723,148.548
C02589=1180.299,296.829,-69.996,-176.792,7.726,148.548
C02590=1180.295,297.077,-70.026,-176.789,7.729,148.548
C02591=1180.290,297.325,-70.056,-176.787,7.732,148.549
C02592=1180.286,297.573,-70.086,-176.785,7.734,148.548
C02593=1180.282,297.822,-70.115,-176.782,7.737,148.548
C02594=1180.277,298.070,-70.146,-176.779,7.740,148.548
C02595=1180.273,298.318,-70.176,-176.777,7.743,148.548
C02596=1180.269,298.565,-70.206,-176.774,7.746,148.549
C02597=1180.265,298.814,-70.236,-176.772,7.749,148.549
C02598=1180.261,299.062,-70.266,-176.769,7.752,148.549
C02599=1180.256,299.310,-70.296,-176.767,7.755,148.548
C02600=1180.252,299.558,-70.326,-176.764,7.758,148.548
C02601=1180.248,299.807,-70.356,-176.762,7.761,148.549
C02602=1180.244,300.055,-70.387,-176.759,7.764,148.549
C02603=1180.239,300.303,-70.416,-176.756,7.767,148.549
C02604=1180.235,300.551,-70.447,-176.754,7.770,148.549
C02605=1180.231,300.799,-70.476,-176.751,7.773,148.549
C02606=1180.227,301.047,-70.507,-176.749,7.775,148.549
C02607=1180.222,301.296,-70.537,-176.747,7.778,148.549
C02608=1180.218,301.543,-70.567,-176.744,7.781,148.549
C02609=1180.214,301.792,-70.598,-176.741,7.784,148.549
C02610=1180.210,302.040,-70.627,-176.738,7.787,148.549
C02611=1180.205,302.288,-70.658,-176.736,7.791,148.549
C02612=1180.201,302.536,-70.688,-176.733,7.794,148.549
C02613=1180.196,302.784,-70.718,-176.731,7.797,148.549
C02614=1180.193,303.032,-70.748,-176.729,7.799,148.549
C02615=1180.189,303.281,-70.780,-176.726,7.802,148.549
C02616=1180.184,303.529,-70.809,-176.724,7.805,148.549
C02617=1180.180,303.777,-70.840,-176.721,7.808,148.549
C02618=1180.175,304.025,-70.871,-176.718,7.811,148.549
C02619=1180.171,304.272,-70.901,-176.716,7.814,148.549
C02620=1180.166,304.521,-70.931,-176.713,7.817,148.549
C02621=1180.163,304.769,-70.961,-176.710,7.820,148.549
C02622=1180.158,305.017,-70.992,-176.708,7.823,148.549
C02623=1180.155,305.265,-71.022,-176.706,7.826,148.549
C02624=1180.150,305.514,-71.052,-176.703,7.829,148.549
C02625=1180.145,305.762,-71.083,-176.700,7.832,148.549
C02626=1180.142,306.010,-71.114,-176.698,7.835,148.549
C02627=1180.137,306.258,-71.144,-176.696,7.838,148.549
C02628=1180.133,306.505,-71.175,-176.693,7.841,148.549
C02629=1180.129,306.753,-71.205,-176.690,7.844,148.549
C02630=1180.125,307.002,-71.236,-176.688,7.847,148.549
C02631=1180.121,307.250,-71.267,-176.685,7.850,148.549
C02632=1180.116,307.498,-71.297,-176.683,7.852,148.549
C02633=1180.111,307.746,-71.327,-176.680,7.855,148.549
C02634=1180.108,307.995,-71.358,-176.678,7.859,148.549
C02635=1180.103,308.243,-71.389,-176.675,7.862,148.549
C02636=1180.099,308.491,-71.420,-176.672,7.865,148.549
C02637=1180.094,308.738,-71.450,-176.670,7.868,148.550
C02638=1180.091,308.987,-71.481,-176.668,7.871,148.550
C02639=1180.086,309.235,-71.512,-176.665,7.874,148.550
C02640=1180.082,309.483,-71.542,-176.663,7.877,148.550
C02641=1180.078,309.731,-71.573,-176.660,7.880,148.550
C02642=1180.074,309.979,-71.604,-176.657,7.883,148.550
C02643=1180.069,310.227,-71.634,-176.655,7.886,148.550
C02644=1180.065,310.476,-71.666,-176.653,7.889,148.550
C02645=1180.062,310.723,-71.696,-176.650,7.892,148.550
C02646=1180.057,310.971,-71.727,-176.647,7.895,148.550
C02647=1180.053,311.219,-71.758,-176.645,7.898,148.550
C02648=1180.048,311.467,-71.789,-176.642,7.901,148.550
C02649=1180.044,311.715,-71.820,-176.640,7.904,148.550
C02650=1180.040,311.964,-71.850,-176.637,7.907,148.550
C02651=1180.036,312.212,-71.881,-176.635,7.910,148.550
C02652=1180.031,312.459,-71.912,-176.632,7.914,148.550
C02653=1180.027,312.708,-71.944,-176.630,7.917,148.550
C02654=1180.023,312.955,-71.975,-176.627,7.920,148.550
C02655=1180.018,313.203,-72.005,-176.625,7.922,148.551
C02656=1180.014,313.452,-72.036,-176.622,7.925,148.551
C02657=1180.011,313.699,-72.067,-176.620,7.928,148.551
C02658=1180.005,313.977,-72.102,-176.617,7.932,148.551
C02659=1180.001,314.253,-72.136,-176.614,7.935,148.551
C02660=1179.996,314.530,-72.172,-176.611,7.938,148.551
C02661=1179.992,314.807,-72.206,-176.609,7.942,148.551
C02662=1179.988,315.054,-72.237,-176.606,7.945,148.551
C02663=1179.983,315.302,-72.268,-176.603,7.948,148.551
C02664=1179.979,315.551,-72.299,-176.601,7.952,148.551
C02665=1179.975,315.798,-72.330,-176.598,7.955,148.551
C02666=1179.971,316.047,-72.362,-176.595,7.958,148.551
C02667=1179.966,316.294,-72.393,-176.594,7.960,148.551
C02668=1179.962,316.543,-72.424,-176.591,7.963,148.551
C02669=1179.958,316.791,-72.455,-176.589,7.967,148.551
C02670=1179.954,317.039,-72.487,-176.586,7.970,148.551
C02671=1179.949,317.287,-72.518,-176.583,7.973,148.551
C02672=1179.945,317.534,-72.549,-176.581,7.976,148.552
C02673=1179.941,317.783,-72.580,-176.578,7.979,148.552
C02674=1179.937,318.030,-72.612,-176.576,7.982,148.552
C02675=1179.933,318.279,-72.643,-176.573,7.985,148.552
C02676=1179.928,318.526,-72.674,-176.571,7.988,148.552
C02677=1179.924,318.775,-72.705,-176.568,7.991,148.552
C02678=1179.920,319.022,-72.737,-176.566,7.994,148.552
C02679=1179.916,319.271,-72.768,-176.563,7.998,148.552
C02680=1179.912,319.518,-72.800,-176.561,8.001,148.552
C02681=1179.908,319.767,-72.831,-176.558,8.004,148.552
C02682=1179.903,320.014,-72.862,-176.556,8.007,148.552
C02683=1179.899,320.263,-72.893,-176.553,8.010,148.553
C02684=1179.896,320.511,-72.925,-176.551,8.013,148.553
C02685=1179.891,320.758,-72.957,-176.548,8.017,148.553
C02686=1179.887,321.007,-72.988,-176.546,8.019,148.553
C02687=1179.883,321.254,-73.019,-176.544,8.022,148.553
C02688=1179.879,321.503,-73.052,-176.541,8.025,148.553
C02689=1179.874,321.751,-73.082,-176.539,8.028,148.553
C02690=1179.870,321.999,-73.114,-176.536,8.031,148.553
C02691=1179.866,322.246,-73.146,-176.534,8.035,148.553
C02692=1179.862,322.495,-73.177,-176.531,8.038,148.553
C02693=1179.858,322.743,-73.209,-176.529,8.041,148.554
C02694=1179.853,322.990,-73.241,-176.526,8.044,148.554
C02695=1179.850,323.238,-73.273,-176.524,8.047,148.554
C02696=1179.845,323.486,-73.303,-176.521,8.050,148.554
C02697=1179.841,323.734,-73.335,-176.519,8.054,148.554
C02698=1179.838,323.982,-73.367,-176.516,8.057,148.554
C02699=1179.833,324.230,-73.399,-176.514,8.060,148.554
C02700=1179.829,324.478,-73.431,-176.511,8.063,148.554
C02701=1179.824,324.726,-73.462,-176.509,8.066,148.554
C02702=1179.820,324.974,-73.494,-176.506,8.069,148.554
C02703=1179.817,325.222,-73.525,-176.504,8.073,148.555
C02704=1179.812,325.470,-73.558,-176.501,8.076,148.555
C02705=1179.808,325.718,-73.589,-176.499,8.079,148.555
C02706=1179.804,325.966,-73.621,-176.496,8.082,148.555
C02707=1179.799,326.213,-73.653,-176.494,8.085,148.555
C02708=1179.796,326.462,-73.685,-176.491,8.088,148.555
C02709=1179.791,326.709,-73.717,-176.489,8.092,148.555
C02710=1179.788,326.957,-73.748,-176.487,8.095,148.555
C02711=1179.783,327.205,-73.781,-176.484,8.098,148.555
C02712=1179.779,327.453,-73.812,-176.482,8.101,148.556
C02713=1179.775,327.701,-73.844,-176.479,8.104,148.556
C02714=1179.771,327.949,-73.877,-176.477,8.107,148.556
C02715=1179.767,328.197,-73.908,-176.474,8.110,148.556
C02716=1179.763,328.444,-73.940,-176.472,8.114,148.556
C02717=1179.758,328.693,-73.972,-176.470,8.117,148.556
C02718=1179.754,328.941,-74.004,-176.467,8.120,148.556
C02719=1179.749,329.188,-74.036,-176.465,8.123,148.556
C02720=1179.746,329.436,-74.068,-176.462,8.126,148.556
C02721=1179.742,329.684,-74.100,-176.460,8.130,148.557
C02722=1179.737,329.932,-74.132,-176.457,8.133,148.557
C02723=1179.733,330.180,-74.164,-176.455,8.136,148.557
C02724=1179.729,330.428,-74.196,-176.452,8.139,148.557
C02725=1179.725,330.677,-74.228,-176.450,8.143,148.557
C02726=1179.720,330.924,-74.261,-176.448,8.146,148.557
C02727=1179.717,331.172,-74.293,-176.445,8.149,148.557
C02728=1179.712,331.420,-74.325,-176.443,8.152,148.558
C02729=1179.709,331.668,-74.357,-176.440,8.155,148.558
C02730=1179.703,331.916,-74.389,-176.438,8.159,148.558
C02731=1179.700,332.163,-74.422,-176.436,8.162,148.558
C02732=1179.696,332.411,-74.454,-176.433,8.165,148.558
C02733=1179.692,332.659,-74.486,-176.431,8.168,148.558
C02734=1179.687,332.907,-74.518,-176.428,8.171,148.558
C02735=1179.683,333.154,-74.551,-176.426,8.174,148.558
C02736=1179.679,333.403,-74.583,-176.424,8.178,148.559
C02737=1179.675,333.651,-74.615,-176.421,8.181,148.559
C02738=1179.671,333.899,-74.648,-176.419,8.184,148.559
C02739=1179.667,334.146,-74.680,-176.416,8.187,148.559
C02740=1179.662,334.394,-74.712,-176.414,8.191,148.559
C02741=1179.659,334.642,-74.745,-176.411,8.194,148.559
C02742=1179.655,334.890,-74.777,-176.409,8.197,148.559
C02743=1179.650,335.138,-74.810,-176.407,8.200,148.560
C02744=1179.646,335.385,-74.842,-176.404,8.204,148.560
C02745=1179.642,335.633,-74.874,-176.402,8.207,148.560
C02746=1179.638,335.881,-74.907,-176.400,8.210,148.560
C02747=1179.634,336.129,-74.939,-176.397,8.213,148.560
C02748=1179.630,336.377,-74.972,-176.395,8.217,148.561
C02749=1179.626,336.625,-75.004,-176.392,8.220,148.561
C02750=1179.622,336.873,-75.037,-176.390,8.223,148.561
C02751=1179.617,337.120,-75.069,-176.388,8.226,148.561
C02752=1179.613,337.368,-75.101,-176.385,8.230,148.561
C02753=1179.609,337.616,-75.134,-176.383,8.233,148.561
C02754=1179.605,337.864,-75.168,-176.380,8.236,148.561
C02755=1179.601,338.112,-75.199,-176.378,8.239,148.562
C02756=1179.597,338.360,-75.233,-176.376,8.242,148.562
C02757=1179.593,338.608,-75.265,-176.374,8.246,148.562
C02758=1179.589,338.855,-75.298,-176.371,8.249,148.562
C02759=1179.585,339.104,-75.330,-176.369,8.252,148.562
C02760=1179.580,339.351,-75.363,-176.366,8.255,148.562
C02761=1179.576,339.599,-75.396,-176.364,8.259,148.563
C02762=1179.572,339.878,-75.432,-176.361,8.263,148.563
C02763=1179.567,340.157,-75.469,-176.359,8.266,148.563
C02764=1179.562,340.436,-75.506,-176.356,8.270,148.563
C02765=1179.558,340.715,-75.543,-176.354,8.273,148.563
C02766=1179.554,340.963,-75.576,-176.351,8.277,148.564
C02767=1179.550,341.211,-75.608,-176.348,8.281,148.564
C02768=1179.545,341.459,-75.642,-176.346,8.284,148.564
C02769=1179.541,341.707,-75.675,-176.344,8.287,148.564
C02770=1179.537,341.954,-75.707,-176.342,8.291,148.565
C02771=1179.533,342.202,-75.739,-176.339,8.294,148.565
C02772=1179.529,342.449,-75.773,-176.337,8.297,148.565
C02773=1179.525,342.697,-75.806,-176.334,8.300,148.565
C02774=1179.520,342.945,-75.839,-176.332,8.304,148.565
C02775=1179.516,343.193,-75.872,-176.330,8.307,148.565
C02776=1179.512,343.441,-75.904,-176.328,8.310,148.566
C02777=1179.508,343.689,-75.938,-176.325,8.314,148.566
C02778=1179.504,343.936,-75.971,-176.323,8.317,148.566
C02779=1179.500,344.184,-76.003,-176.321,8.320,148.566
C02780=1179.496,344.432,-76.036,-176.319,8.323,148.566
C02781=1179.492,344.679,-76.070,-176.316,8.327,148.567
C02782=1179.488,344.927,-76.103,-176.314,8.330,148.567
C02783=1179.484,345.175,-76.136,-176.312,8.333,148.567
C02784=1179.479,345.423,-76.169,-176.309,8.337,148.567
C02785=1179.475,345.671,-76.202,-176.307,8.340,148.568
C02786=1179.471,345.919,-76.235,-176.304,8.344,148.568
C02787=1179.467,346.166,-76.268,-176.302,8.347,148.568
C02788=1179.463,346.414,-76.301,-176.300,8.351,148.568
C02789=1179.459,346.662,-76.334,-176.298,8.354,148.568
C02790=1179.455,346.910,-76.368,-176.295,8.357,148.569
C02791=1179.451,347.158,-76.401,-176.293,8.361,148.569
C02792=1179.447,347.406,-76.434,-176.291,8.364,148.569
C02793=1179.443,347.653,-76.468,-176.289,8.367,148.569
C02794=1179.439,347.901,-76.501,-176.286,8.371,148.570
C02795=1179.435,348.148,-76.534,-176.284,8.374,148.570
C02796=1179.430,348.396,-76.567,-176.282,8.377,148.570
C02797=1179.426,348.644,-76.600,-176.279,8.381,148.570
C02798=1179.422,348.891,-76.634,-176.277,8.384,148.570
C02799=1179.418,349.139,-76.667,-176.275,8.387,148.571
C02800=1179.414,349.387,-76.700,-176.272,8.391,148.571
C02801=1179.410,349.635,-76.733,-176.270,8.395,148.571
C02802=1179.407,349.882,-76.767,-176.268,8.398,148.572
C02803=1179.402,350.130,-76.801,-176.266,8.402,148.572
C02804=1179.397,350.378,-76.834,-176.263,8.405,148.572
C02805=1179.393,350.626,-76.867,-176.261,8.408,148.572
C02806=1179.389,350.874,-76.901,-176.259,8.412,148.572
C02807=1179.385,351.121,-76.934,-176.257,8.415,148.573
C02808=1179.381,351.368,-76.968,-176.255,8.418,148.573
C02809=1179.378,351.617,-77.001,-176.253,8.422,148.573
C02810=1179.374,351.865,-77.034,-176.250,8.425,148.573
C02811=1179.369,352.112,-77.069,-176.248,8.428,148.574
C02812=1179.365,352.360,-77.102,-176.245,8.433,148.574
C02813=1179.361,352.608,-77.135,-176.243,8.436,148.574
C02814=1179.357,352.855,-77.169,-176.241,8.439,148.575
C02815=1179.353,353.103,-77.202,-176.239,8.443,148.575
C02816=1179.349,353.351,-77.236,-176.237,8.446,148.575
C02817=1179.345,353.598,-77.270,-176.234,8.449,148.575
C02818=1179.341,353.846,-77.303,-176.233,8.453,148.576
C02819=1179.337,354.093,-77.337,-176.230,8.456,148.576
C02820=1179.333,354.341,-77.371,-176.228,8.460,148.576
C02821=1179.328,354.590,-77.404,-176.226,8.463,148.576
C02822=1179.324,354.837,-77.438,-176.223,8.467,148.577
C02823=1179.320,355.084,-77.471,-176.221,8.471,148.577
C02824=1179.316,355.331,-77.505,-176.219,8.474,148.577
C02825=1179.312,355.580,-77.539,-176.217,8.478,148.578
C02826=1179.308,355.827,-77.573,-176.215,8.481,148.578
C02827=1179.304,356.075,-77.606,-176.212,8.484,148.578
C02828=1179.300,356.322,-77.640,-176.211,8.488,148.579
C02829=1179.296,356.571,-77.674,-176.208,8.491,148.579
C02830=1179.292,356.818,-77.708,-176.206,8.494,148.579
C02831=1179.288,357.066,-77.741,-176.204,8.498,148.579
C02832=1179.284,357.313,-77.776,-176.201,8.502,148.580
C02833=1179.280,357.562,-77.809,-176.199,8.506,148.580
C02834=1179.276,357.809,-77.843,-176.197,8.509,148.580
C02835=1179.272,358.056,-77.878,-176.195,8.512,148.581
C02836=1179.268,358.305,-77.911,-176.193,8.516,148.581
C02837=1179.264,358.552,-77.945,-176.191,8.519,148.581
C02838=1179.260,358.799,-77.980,-176.189,8.523,148.582
C02839=1179.256,359.048,-78.013,-176.187,8.526,148.582
C02840=1179.252,359.295,-78.048,-176.185,8.530,148.582
C02841=1179.248,359.542,-78.081,-176.182,8.534,148.583
C02842=1179.244,359.790,-78.115,-176.180,8.538,148.583
C02843=1179.240,360.038,-78.149,-176.178,8.541,148.583
C02844=1179.236,360.285,-78.183,-176.176,8.545,148.584
C02845=1179.231,360.533,-78.217,-176.174,8.548,148.584
C02846=1179.228,360.781,-78.251,-176.172,8.552,148.584
C02847=1179.223,361.028,-78.286,-176.170,8.555,148.585
C02848=1179.219,361.275,-78.320,-176.168,8.558,148.585
C02849=1179.216,361.523,-78.354,-176.166,8.562,148.585
C02850=1179.211,361.771,-78.388,-176.164,8.565,148.586
C02851=1179.208,362.019,-78.422,-176.162,8.569,148.586
C02852=1179.203,362.266,-78.456,-176.160,8.573,148.587
C02853=1179.200,362.514,-78.490,-176.158,8.576,148.587
C02854=1179.196,362.762,-78.525,-176.156,8.580,148.587
C02855=1179.192,363.009,-78.559,-176.154,8.583,148.588
C02856=1179.187,363.257,-78.593,-176.152,8.586,148.588
C02857=1179.184,363.505,-78.627,-176.150,8.590,148.588
C02858=1179.179,363.752,-78.661,-176.149,8.594,148.589
C02859=1179.176,364.000,-78.696,-176.147,8.597,148.589
C02860=1179.171,364.247,-78.730,-176.145,8.601,148.590
C02861=1179.167,364.494,-78.764,-176.143,8.604,148.590
C02862=1179.163,364.743,-78.799,-176.141,8.608,148.590
C02863=1179.159,364.990,-78.833,-176.139,8.612,148.591
C02864=1179.156,365.238,-78.867,-176.137,8.615,148.591
C02865=1179.151,365.485,-78.902,-176.135,8.619,148.592
C02866=1179.147,365.766,-78.941,-176.133,8.623,148.592
C02867=1179.142,366.048,-78.980,-176.131,8.627,148.592
C02868=1179.138,366.331,-79.019,-176.129,8.631,148.593
C02869=1179.133,366.612,-79.058,-176.127,8.635,148.593
C02870=1179.129,366.860,-79.093,-176.125,8.638,148.594
C02871=1179.126,367.108,-79.127,-176.123,8.642,148.594
C02872=1179.121,367.355,-79.161,-176.121,8.646,148.595
C02873=1179.117,367.602,-79.197,-176.120,8.649,148.595
C02874=1179.114,367.850,-79.231,-176.118,8.653,148.596
C02875=1179.109,368.097,-79.265,-176.116,8.657,148.596
C02876=1179.105,368.345,-79.300,-176.115,8.660,148.597
C02877=1179.101,368.592,-79.334,-176.113,8.664,148.597
C02878=1179.097,368.840,-79.369,-176.111,8.667,148.597
C02879=1179.093,369.088,-79.403,-176.110,8.671,148.598
C02880=1179.090,369.335,-79.438,-176.108,8.674,148.598
C02881=1179.085,369.582,-79.473,-176.106,8.678,148.599
C02882=1179.081,369.831,-79.507,-176.105,8.682,148.599
C02883=1179.077,370.078,-79.542,-176.103,8.685,148.600
C02884=1179.073,370.326,-79.576,-176.102,8.688,148.600
C02885=1179.069,370.573,-79.611,-176.100,8.692,148.601
C02886=1179.065,370.821,-79.646,-176.098,8.696,148.601
C02887=1179.061,371.068,-79.681,-176.096,8.699,148.602
C02888=1179.057,371.316,-79.715,-176.096,8.702,148.602
C02889=1179.053,371.563,-79.750,-176.094,8.706,148.603
C02890=1179.049,371.811,-79.785,-176.092,8.710,148.603
C02891=1179.045,372.058,-79.819,-176.091,8.713,148.604
C02892=1179.041,372.306,-79.854,-176.089,8.716,148.604
C02893=1179.038,372.554,-79.889,-176.088,8.720,148.605
C02894=1179.033,372.801,-79.924,-176.086,8.724,148.605
C02895=1179.029,373.049,-79.958,-176.085,8.728,148.606
C02896=1179.025,373.296,-79.994,-176.084,8.730,148.606
C02897=1179.022,373.544,-80.028,-176.082,8.734,148.607
C02898=1179.017,373.791,-80.063,-176.080,8.738,148.607
C02899=1179.013,374.039,-80.098,-176.079,8.741,148.608
C02900=1179.009,374.287,-80.133,-176.078,8.745,148.608
C02901=1179.005,374.534,-80.168,-176.077,8.748,148.609
C02902=1179.001,374.782,-80.203,-176.075,8.752,148.609
C02903=1178.998,375.028,-80.237,-176.074,8.755,148.610
C02904=1178.994,375.276,-80.272,-176.073,8.758,148.610
C02905=1178.989,375.524,-80.307,-176.071,8.762,148.611
C02906=1178.985,375.771,-80.342,-176.071,8.765,148.612
C02907=1178.981,376.019,-80.377,-176.069,8.769,148.612
C02908=1178.977,376.266,-80.412,-176.068,8.772,148.613
C02909=1178.973,376.514,-80.447,-176.067,8.776,148.613
C02910=1178.969,376.761,-80.482,-176.066,8.779,148.614
C02911=1178.965,377.009,-80.517,-176.064,8.783,148.614
C02912=1178.962,377.256,-80.552,-176.063,8.786,148.615
C02913=1178.957,377.504,-80.586,-176.062,8.790,148.616
C02914=1178.954,377.751,-80.622,-176.061,8.793,148.616
C02915=1178.950,377.999,-80.657,-176.059,8.797,148.617
C02916=1178.946,378.246,-80.692,-176.059,8.800,148.617
C02917=1178.942,378.494,-80.728,-176.057,8.804,148.618
C02918=1178.937,378.741,-80.762,-176.056,8.807,148.618
C02919=1178.934,378.989,-80.798,-176.055,8.810,148.619
C02920=1178.930,379.237,-80.832,-176.054,8.814,148.620
C02921=1178.925,379.484,-80.868,-176.053,8.817,148.620
C02922=1178.922,379.731,-80.903,-176.052,8.820,148.621
C02923=1178.918,379.979,-80.938,-176.051,8.824,148.621
C02924=1178.914,380.226,-80.973,-176.050,8.827,148.622
C02925=1178.910,380.474,-81.008,-176.049,8.830,148.623
C02926=1178.906,380.722,-81.044,-176.048,8.833,148.623
C02927=1178.902,380.968,-81.079,-176.047,8.837,148.624
C02928=1178.898,381.217,-81.114,-176.046,8.840,148.624
C02929=1178.894,381.464,-81.149,-176.045,8.843,148.625
C02930=1178.890,381.711,-81.184,-176.045,8.847,148.626
C02931=1178.886,381.959,-81.219,-176.044,8.850,148.626
C02932=1178.882,382.206,-81.255,-176.043,8.854,148.627
C02933=1178.878,382.453,-81.290,-176.042,8.857,148.627
C02934=1178.874,382.701,-81.325,-176.041,8.860,148.628
C02935=1178.870,382.949,-81.360,-176.040,8.863,148.629
C02936=1178.866,383.196,-81.395,-176.040,8.866,148.629
C02937=1178.862,383.443,-81.431,-176.039,8.869,148.630
C02938=1178.859,383.691,-81.467,-176.038,8.872,148.631
C02939=1178.855,383.939,-81.501,-176.037,8.875,148.631
C02940=1178.850,384.186,-81.537,-176.037,8.879,148.632
C02941=1178.846,384.433,-81.573,-176.036,8.882,148.632
C02942=1178.842,384.681,-81.608,-176.035,8.885,148.633
C02943=1178.838,384.928,-81.643,-176.034,8.888,148.634
C02944=1178.834,385.176,-81.678,-176.034,8.892,148.634
C02945=1178.830,385.423,-81.714,-176.033,8.895,148.635
C02946=1178.827,385.671,-81.749,-176.032,8.898,148.636
C02947=1178.823,385.918,-81.785,-176.032,8.901,148.636
C02948=1178.819,386.165,-81.820,-176.031,8.904,148.637
C02949=1178.815,386.413,-81.855,-176.031,8.907,148.638
C02950=1178.811,386.661,-81.890,-176.030,8.910,148.638
C02951=1178.806,386.908,-81.926,-176.030,8.913,148.639
C02952=1178.803,387.155,-81.962,-176.029,8.916,148.640
C02953=1178.799,387.403,-81.997,-176.028,8.919,148.640
C02954=1178.795,387.650,-82.033,-176.029,8.922,148.641
C02955=1178.791,387.897,-82.068,-176.028,8.925,148.641
C02956=1178.787,388.145,-82.103,-176.027,8.929,148.642
C02957=1178.783,388.393,-82.138,-176.027,8.931,148.643
C02958=1178.779,388.641,-82.175,-176.027,8.934,148.644
C02959=1178.775,388.887,-82.210,-176.026,8.937,148.644
C02960=1178.771,389.135,-82.245,-176.026,8.940,148.645
C02961=1178.767,389.382,-82.281,-176.025,8.943,148.645
C02962=1178.764,389.630,-82.316,-176.025,8.945,148.646
C02963=1178.759,389.877,-82.352,-176.025,8.949,148.647
C02964=1178.755,390.125,-82.388,-176.024,8.952,148.648
C02965=1178.751,390.372,-82.423,-176.024,8.955,148.648
C02966=1178.748,390.620,-82.459,-176.024,8.958,148.649
C02967=1178.744,390.867,-82.494,-176.024,8.960,148.650
C02968=1178.740,391.114,-82.530,-176.023,8.962,148.650
C02969=1178.736,391.361,-82.565,-176.023,8.966,148.651
C02970=1178.731,391.646,-82.606,-176.023,8.969,148.652
C02971=1178.727,391.930,-82.647,-176.022,8.973,148.652
C02972=1178.722,392.215,-82.688,-176.022,8.975,148.653
C02973=1178.718,392.499,-82.729,-176.022,8.979,148.654
C02974=1178.714,392.746,-82.764,-176.022,8.981,148.654
C02975=1178.710,392.993,-82.800,-176.021,8.984,148.655
C02976=1178.706,393.241,-82.836,-176.022,8.987,148.656
C02977=1178.702,393.488,-82.871,-176.021,8.989,148.656
C02978=1178.699,393.736,-82.907,-176.021,8.993,148.657
C02979=1178.694,393.983,-82.942,-176.021,8.995,148.658
C02980=1178.690,394.231,-82.978,-176.021,8.997,148.658
C02981=1178.686,394.478,-83.014,-176.021,9.000,148.659
C02982=1178.683,394.726,-83.049,-176.021,9.003,148.660
C02983=1178.679,394.973,-83.085,-176.020,9.006,148.660
C02984=1178.674,395.220,-83.121,-176.020,9.008,148.661
C02985=1178.670,395.468,-83.156,-176.020,9.010,148.662
C02986=1178.667,395.715,-83.192,-176.020,9.013,148.662
C02987=1178.663,395.963,-83.227,-176.020,9.016,148.663
C02988=1178.658,396.210,-83.264,-176.020,9.019,148.664
C02989=1178.654,396.457,-83.299,-176.020,9.021,148.664
C02990=1178.651,396.705,-83.334,-176.020,9.024,148.665
C02991=1178.646,396.953,-83.370,-176.020,9.026,148.666
C02992=1178.643,397.199,-83.407,-176.020,9.029,148.666
C02993=1178.639,397.447,-83.442,-176.020,9.031,148.667
C02994=1178.635,397.694,-83.478,-176.020,9.033,148.668
C02995=1178.630,397.942,-83.514,-176.020,9.036,148.668
C02996=1178.627,398.189,-83.549,-176.020,9.039,148.669
C02997=1178.623,398.437,-83.585,-176.020,9.041,148.670
C02998=1178.619,398.684,-83.621,-176.020,9.043,148.670
C02999=1178.615,398.932,-83.656,-176.020,9.046,148.671
C03000=1178.611,399.179,-83.692,-176.020,9.048,148.672
C03001=1178.607,399.426,-83.728,-176.020,9.051,148.672
C03002=1178.603,399.673,-83.764,-176.020,9.053,148.673
C03003=1178.599,399.921,-83.800,-176.020,9.056,148.674
C03004=1178.596,400.168,-83.835,-176.020,9.058,148.674
C03005=1178.591,400.416,-83.871,-176.020,9.060,148.675
C03006=1178.588,400.664,-83.907,-176.020,9.063,148.675
C03007=1178.584,400.911,-83.943,-176.020,9.065,148.676
C03008=1178.579,401.158,-83.979,-176.020,9.068,148.677
C03009=1178.576,401.405,-84.014,-176.020,9.070,148.677
C03010=1178.572,401.653,-84.050,-176.020,9.072,148.678
C03011=1178.568,401.901,-84.086,-176.021,9.074,148.679
C03012=1178.564,402.148,-84.122,-176.020,9.077,148.679
C03013=1178.561,402.395,-84.158,-176.021,9.079,148.680
C03014=1178.556,402.643,-84.194,-176.020,9.082,148.680
C03015=1178.552,402.889,-84.229,-176.020,9.084,148.681
C03016=1178.548,403.137,-84.265,-176.021,9.086,148.682
C03017=1178.544,403.385,-84.301,-176.021,9.088,148.682
C03018=1178.540,403.632,-84.337,-176.021,9.091,148.683
C03019=1178.537,403.879,-84.373,-176.021,9.093,148.683
C03020=1178.532,404.127,-84.409,-176.022,9.095,148.684
C03021=1178.529,404.375,-84.444,-176.021,9.097,148.685
C03022=1178.524,404.621,-84.480,-176.021,9.099,148.685
C03023=1178.520,404.868,-84.516,-176.021,9.102,148.686
C03024=1178.517,405.116,-84.552,-176.022,9.104,148.687
C03025=1178.513,405.363,-84.587,-176.022,9.106,148.687
C03026=1178.509,405.611,-84.624,-176.022,9.108,148.688
C03027=1178.505,405.858,-84.660,-176.021,9.111,148.688
C03028=1178.501,406.106,-84.696,-176.022,9.112,148.689
C03029=1178.497,406.353,-84.732,-176.022,9.115,148.690
C03030=1178.494,406.601,-84.767,-176.022,9.117,148.690
C03031=1178.489,406.847,-84.804,-176.022,9.119,148.691
C03032=1178.485,407.095,-84.839,-176.023,9.121,148.691
C03033=1178.482,407.342,-84.875,-176.023,9.123,148.692
C03034=1178.477,407.590,-84.911,-176.023,9.125,148.693
C03035=1178.474,407.837,-84.947,-176.023,9.127,148.693
C03036=1178.469,408.085,-84.983,-176.024,9.129,148.694
C03037=1178.466,408.332,-85.019,-176.023,9.131,148.694
C03038=1178.462,408.579,-85.055,-176.023,9.134,148.695
C03039=1178.458,408.827,-85.091,-176.024,9.135,148.695
C03040=1178.454,409.074,-85.126,-176.023,9.138,148.696
C03041=1178.450,409.321,-85.162,-176.024,9.139,148.697
C03042=1178.446,409.569,-85.199,-176.024,9.142,148.697
C03043=1178.442,409.816,-85.234,-176.024,9.143,148.698
C03044=1178.438,410.064,-85.270,-176.024,9.146,148.698
C03045=1178.435,410.311,-85.307,-176.024,9.148,148.699
C03046=1178.431,410.558,-85.342,-176.024,9.149,148.699
C03047=1178.426,410.806,-85.378,-176.025,9.152,148.700
C03048=1178.423,411.053,-85.415,-176.025,9.153,148.700
C03049=1178.419,411.301,-85.451,-176.025,9.156,148.701
C03050=1178.414,411.548,-85.486,-176.025,9.157,148.702
C03051=1178.411,411.795,-85.522,-176.025,9.160,148.702
C03052=1178.407,412.042,-85.558,-176.025,9.161,148.703
C03053=1178.403,412.290,-85.594,-176.025,9.164,148.703
C03054=1178.399,412.538,-85.630,-176.026,9.165,148.704
C03055=1178.395,412.785,-85.666,-176.025,9.167,148.704
C03056=1178.391,413.032,-85.703,-176.026,9.169,148.705
C03057=1178.387,413.280,-85.738,-176.026,9.171,148.705
C03058=1178.384,413.527,-85.774,-176.026,9.173,148.706
C03059=1178.379,413.775,-85.810,-176.026,9.175,148.706
C03060=1178.376,414.021,-85.847,-176.027,9.177,148.707
C03061=1178.372,414.269,-85.883,-176.026,9.179,148.708
C03062=1178.367,414.516,-85.918,-176.027,9.181,148.708
C03063=1178.363,414.763,-85.955,-176.026,9.183,148.709
C03064=1178.360,415.011,-85.990,-176.027,9.185,148.709
C03065=1178.355,415.259,-86.027,-176.027,9.187,148.710
C03066=1178.353,415.494,-86.061,-176.027,9.188,148.710
C03067=1178.349,415.731,-86.096,-176.027,9.190,148.711
C03068=1178.346,415.968,-86.130,-176.027,9.192,148.711
C03069=1178.345,416.204,-86.164,-176.027,9.193,148.712
C03070=1178.344,416.440,-86.198,-176.028,9.195,148.712
C03071=1178.345,416.676,-86.232,-176.027,9.197,148.713
C03072=1178.346,416.912,-86.266,-176.028,9.199,148.713
C03073=1178.349,417.148,-86.299,-176.028,9.200,148.713
C03074=1177.928,417.148,-86.343,-176.031,9.211,148.717
C03075=1177.926,416.911,-86.309,-176.031,9.209,148.717
C03076=1177.924,416.674,-86.275,-176.030,9.208,148.716
C03077=1177.923,416.437,-86.241,-176.031,9.205,148.716
C03078=1177.923,416.198,-86.206,-176.030,9.204,148.715
C03079=1177.925,415.960,-86.172,-176.030,9.203,148.715
C03080=1177.927,415.723,-86.137,-176.030,9.200,148.714
C03081=1177.931,415.485,-86.103,-176.030,9.199,148.714
C03082=1177.934,415.247,-86.068,-176.030,9.197,148.713
C03083=1177.939,415.000,-86.032,-176.030,9.195,148.713
C03084=1177.943,414.752,-85.996,-176.030,9.194,148.712
C03085=1177.946,414.505,-85.960,-176.030,9.192,148.712
C03086=1177.950,414.257,-85.924,-176.029,9.190,148.711
C03087=1177.954,414.010,-85.887,-176.030,9.188,148.711
C03088=1177.959,413.763,-85.852,-176.029,9.186,148.710
C03089=1177.962,413.516,-85.816,-176.030,9.184,148.710
C03090=1177.966,413.269,-85.779,-176.029,9.182,148.709
C03091=1177.970,413.021,-85.744,-176.029,9.180,148.709
C03092=1177.974,412.773,-85.708,-176.029,9.178,148.708
C03093=1177.978,412.526,-85.671,-176.029,9.176,148.707
C03094=1177.981,412.279,-85.636,-176.028,9.174,148.707
C03095=1177.986,412.031,-85.600,-176.029,9.172,148.706
C03096=1177.989,411.784,-85.563,-176.028,9.170,148.706
C03097=1177.994,411.536,-85.527,-176.028,9.168,148.705
C03098=1177.997,411.289,-85.492,-176.028,9.167,148.705
C03099=1178.001,411.042,-85.455,-176.028,9.164,148.704
C03100=1178.006,410.795,-85.420,-176.027,9.163,148.704
C03101=1178.009,410.547,-85.384,-176.028,9.160,148.703
C03102=1178.013,410.300,-85.347,-176.027,9.159,148.702
C03103=1178.017,410.053,-85.312,-176.027,9.156,148.702
C03104=1178.021,409.805,-85.275,-176.027,9.155,148.701
C03105=1178.025,409.558,-85.239,-176.027,9.152,148.701
C03106=1178.029,409.311,-85.204,-176.027,9.151,148.700
C03107=1178.033,409.063,-85.168,-176.026,9.148,148.700
C03108=1178.036,408.816,-85.131,-176.027,9.146,148.699
C03109=1178.041,408.568,-85.095,-176.026,9.145,148.699
C03110=1178.044,408.321,-85.060,-176.026,9.142,148.698
C03111=1178.049,408.074,-85.024,-176.026,9.141,148.697
C03112=1178.053,407.827,-84.988,-176.026,9.138,148.697
C03113=1178.056,407.579,-84.952,-176.026,9.136,148.696
C03114=1178.060,407.332,-84.916,-176.025,9.134,148.696
C03115=1178.064,407.084,-84.880,-176.026,9.132,148.695
C03116=1178.068,406.837,-84.844,-176.025,9.130,148.694
C03117=1178.072,406.589,-84.808,-176.025,9.128,148.694
C03118=1178.076,406.342,-84.772,-176.025,9.125,148.693
C03119=1178.079,406.095,-84.736,-176.025,9.124,148.693
C03120=1178.084,405.848,-84.700,-176.024,9.121,148.692
C03121=1178.088,405.600,-84.665,-176.025,9.119,148.691
C03122=1178.092,405.353,-84.629,-176.024,9.117,148.691
C03123=1178.096,405.105,-84.592,-176.024,9.115,148.690
C03124=1178.099,404.858,-84.557,-176.024,9.112,148.690
C03125=1178.104,404.610,-84.521,-176.024,9.110,148.689
C03126=1178.107,404.363,-84.485,-176.024,9.108,148.688
C03127=1178.111,404.116,-84.449,-176.024,9.106,148.688
C03128=1178.115,403.868,-84.413,-176.024,9.104,148.687
C03129=1178.119,403.621,-84.378,-176.024,9.101,148.687
C03130=1178.123,403.374,-84.342,-176.023,9.100,148.686
C03131=1178.127,403.126,-84.306,-176.023,9.097,148.685
C03132=1178.131,402.879,-84.270,-176.023,9.095,148.685
C03133=1178.134,402.631,-84.234,-176.023,9.092,148.684
C03134=1178.139,402.384,-84.198,-176.023,9.091,148.684
C03135=1178.143,402.136,-84.162,-176.023,9.088,148.683
C03136=1178.147,401.889,-84.127,-176.023,9.086,148.682
C03137=1178.151,401.642,-84.090,-176.023,9.083,148.682
C03138=1178.155,401.395,-84.055,-176.023,9.081,148.681
C03139=1178.158,401.147,-84.019,-176.023,9.079,148.680
C03140=1178.163,400.899,-83.983,-176.023,9.076,148.680
C03141=1178.166,400.652,-83.948,-176.022,9.074,148.679
C03142=1178.170,400.405,-83.911,-176.022,9.072,148.678
C03143=1178.175,400.158,-83.875,-176.022,9.069,148.678
C03144=1178.178,399.910,-83.840,-176.022,9.067,148.677
C03145=1178.182,399.663,-83.804,-176.022,9.065,148.676
C03146=1178.186,399.415,-83.768,-176.022,9.062,148.676
C03147=1178.190,399.167,-83.733,-176.022,9.060,148.675
C03148=1178.194,398.920,-83.697,-176.022,9.057,148.675
C03149=1178.198,398.673,-83.660,-176.022,9.055,148.674
C03150=1178.202,398.426,-83.625,-176.022,9.052,148.673
C03151=1178.206,398.179,-83.590,-176.022,9.050,148.673
C03152=1178.209,397.931,-83.554,-176.022,9.047,148.672
C03153=1178.214,397.683,-83.518,-176.022,9.045,148.671
C03154=1178.217,397.436,-83.482,-176.022,9.042,148.671
C03155=1178.221,397.188,-83.447,-176.022,9.040,148.670
C03156=1178.226,396.941,-83.411,-176.022,9.038,148.669
C03157=1178.229,396.694,-83.375,-176.022,9.035,148.669
C03158=1178.233,396.447,-83.339,-176.022,9.032,148.668
C03159=1178.237,396.199,-83.304,-176.023,9.029,148.667
C03160=1178.241,395.951,-83.267,-176.023,9.027,148.667
C03161=1178.245,395.704,-83.232,-176.022,9.024,148.666
C03162=1178.249,395.457,-83.197,-176.023,9.022,148.665
C03163=1178.253,395.209,-83.161,-176.022,9.019,148.665
C03164=1178.257,394.962,-83.125,-176.023,9.017,148.664
C03165=1178.261,394.714,-83.090,-176.023,9.014,148.663
C03166=1178.264,394.467,-83.054,-176.023,9.011,148.663
C03167=1178.269,394.220,-83.018,-176.023,9.009,148.662
C03168=1178.273,393.972,-82.983,-176.023,9.006,148.661
C03169=1178.277,393.725,-82.947,-176.023,9.003,148.661
C03170=1178.280,393.478,-82.911,-176.024,9.001,148.660
C03171=1178.285,393.230,-82.875,-176.024,8.998,148.659
C03172=1178.289,392.983,-82.840,-176.023,8.995,148.659
C03173=1178.292,392.736,-82.804,-176.024,8.992,148.658
C03174=1178.296,392.488,-82.768,-176.024,8.990,148.657
C03175=1178.301,392.203,-82.727,-176.024,8.986,148.657
C03176=1178.305,391.920,-82.687,-176.025,8.983,148.656
C03177=1178.310,391.635,-82.646,-176.025,8.980,148.655
C03178=1178.314,391.351,-82.604,-176.025,8.977,148.654
C03179=1178.318,391.104,-82.569,-176.025,8.974,148.654
C03180=1178.322,390.856,-82.534,-176.026,8.971,148.653
C03181=1178.326,390.609,-82.498,-176.026,8.968,148.652
C03182=1178.330,390.360,-82.463,-176.026,8.966,148.652
C03183=1178.334,390.113,-82.427,-176.027,8.962,148.651
C03184=1178.338,389.866,-82.392,-176.027,8.960,148.650
C03185=1178.342,389.619,-82.356,-176.027,8.957,148.650
C03186=1178.346,389.371,-82.321,-176.027,8.954,148.649
C03187=1178.350,389.123,-82.285,-176.028,8.951,148.648
C03188=1178.354,388.877,-82.250,-176.028,8.948,148.648
C03189=1178.358,388.629,-82.214,-176.029,8.945,148.647
C03190=1178.362,388.382,-82.178,-176.029,8.942,148.646
C03191=1178.365,388.134,-82.143,-176.029,8.940,148.646
C03192=1178.370,387.887,-82.108,-176.030,8.936,148.645
C03193=1178.374,387.639,-82.072,-176.031,8.933,148.644
C03194=1178.378,387.392,-82.036,-176.031,8.930,148.644
C03195=1178.382,387.144,-82.001,-176.031,8.928,148.643
C03196=1178.385,386.896,-81.966,-176.032,8.924,148.642
C03197=1178.390,386.649,-81.931,-176.032,8.921,148.642
C03198=1178.393,386.402,-81.895,-176.033,8.918,148.641
C03199=1178.397,386.154,-81.859,-176.034,8.915,148.640
C03200=1178.401,385.908,-81.824,-176.034,8.912,148.640
C03201=1178.406,385.660,-81.788,-176.034,8.909,148.639
C03202=1178.409,385.412,-81.753,-176.035,8.906,148.639
C03203=1178.413,385.164,-81.718,-176.036,8.902,148.638
C03204=1178.417,384.917,-81.683,-176.036,8.899,148.637
C03205=1178.421,384.670,-81.647,-176.037,8.896,148.637
C03206=1178.425,384.422,-81.611,-176.038,8.893,148.636
C03207=1178.428,384.175,-81.576,-176.038,8.890,148.635
C03208=1178.433,383.928,-81.541,-176.039,8.887,148.635
C03209=1178.437,383.680,-81.506,-176.040,8.884,148.634
C03210=1178.440,383.433,-81.470,-176.041,8.880,148.633
C03211=1178.445,383.186,-81.435,-176.041,8.877,148.633
C03212=1178.449,382.938,-81.400,-176.042,8.874,148.632
C03213=1178.453,382.690,-81.364,-176.043,8.871,148.632
C03214=1178.457,382.442,-81.329,-176.043,8.868,148.631
C03215=1178.461,382.196,-81.293,-176.045,8.864,148.630
C03216=1178.465,381.947,-81.259,-176.046,8.861,148.630
C03217=1178.468,381.700,-81.223,-176.046,8.857,148.629
C03218=1178.473,381.453,-81.188,-176.047,8.854,148.628
C03219=1178.477,381.205,-81.153,-176.048,8.851,148.628
C03220=1178.480,380.957,-81.117,-176.049,8.847,148.627
C03221=1178.485,380.711,-81.082,-176.050,8.844,148.627
C03222=1178.489,380.463,-81.047,-176.051,8.841,148.626
C03223=1178.492,380.215,-81.012,-176.052,8.838,148.625
C03224=1178.497,379.968,-80.977,-176.053,8.834,148.625
C03225=1178.501,379.720,-80.942,-176.054,8.831,148.624
C03226=1178.504,379.473,-80.906,-176.055,8.828,148.623
C03227=1178.508,379.226,-80.871,-176.056,8.824,148.623
C03228=1178.512,378.978,-80.836,-176.057,8.821,148.622
C03229=1178.516,378.730,-80.801,-176.058,8.818,148.622
C03230=1178.521,378.483,-80.766,-176.059,8.814,148.621
C03231=1178.524,378.235,-80.731,-176.060,8.811,148.621
C03232=1178.529,377.988,-80.696,-176.062,8.807,148.620
C03233=1178.533,377.740,-80.661,-176.062,8.804,148.619
C03234=1178.536,377.493,-80.625,-176.063,8.801,148.619
C03235=1178.540,377.246,-80.591,-176.065,8.797,148.618
C03236=1178.544,376.998,-80.556,-176.066,8.794,148.618
C03237=1178.548,376.750,-80.521,-176.067,8.790,148.617
C03238=1178.552,376.503,-80.486,-176.068,8.787,148.617
C03239=1178.556,376.255,-80.451,-176.070,8.783,148.616
C03240=1178.560,376.008,-80.416,-176.070,8.780,148.615
C03241=1178.564,375.760,-80.381,-176.072,8.776,148.615
C03242=1178.568,375.513,-80.345,-176.074,8.772,148.614
C03243=1178.572,375.265,-80.311,-176.074,8.769,148.614
C03244=1178.576,375.018,-80.275,-176.076,8.766,148.613
C03245=1178.580,374.771,-80.242,-176.077,8.763,148.613
C03246=1178.584,374.523,-80.207,-176.078,8.759,148.612
C03247=1178.587,374.275,-80.171,-176.080,8.755,148.612
C03248=1178.592,374.028,-80.137,-176.081,8.752,148.611
C03249=1178.596,373.780,-80.101,-176.083,8.748,148.611
C03250=1178.600,373.533,-80.067,-176.084,8.745,148.610
C03251=1178.604,373.285,-80.032,-176.086,8.742,148.610
C03252=1178.608,373.038,-79.997,-176.087,8.738,148.609
C03253=1178.612,372.790,-79.962,-176.088,8.734,148.608
C03254=1178.616,372.542,-79.928,-176.090,8.731,148.608
C03255=1178.620,372.295,-79.892,-176.091,8.727,148.608
C03256=1178.623,372.047,-79.858,-176.093,8.724,148.607
C03257=1178.628,371.800,-79.824,-176.095,8.720,148.607
C03258=1178.631,371.552,-79.788,-176.096,8.717,148.606
C03259=1178.636,371.305,-79.754,-176.097,8.713,148.605
C03260=1178.640,371.057,-79.719,-176.099,8.710,148.605
C03261=1178.644,370.810,-79.684,-176.101,8.706,148.604
C03262=1178.647,370.562,-79.649,-176.102,8.703,148.604
C03263=1178.652,370.315,-79.615,-176.104,8.699,148.604
C03264=1178.656,370.067,-79.580,-176.105,8.695,148.603
C03265=1178.660,369.820,-79.546,-176.107,8.692,148.603
C03266=1178.664,369.572,-79.511,-176.109,8.688,148.602
C03267=1178.668,369.325,-79.476,-176.111,8.685,148.602
C03268=1178.671,369.077,-79.442,-176.111,8.681,148.601
C03269=1178.676,368.829,-79.408,-176.113,8.678,148.601
C03270=1178.680,368.581,-79.373,-176.115,8.674,148.600
C03271=1178.684,368.335,-79.338,-176.117,8.671,148.600
C03272=1178.687,368.087,-79.303,-176.119,8.667,148.599
C03273=1178.692,367.839,-79.269,-176.120,8.663,148.599
C03274=1178.696,367.591,-79.234,-176.122,8.660,148.599
C03275=1178.700,367.344,-79.200,-176.124,8.656,148.598
C03276=1178.704,367.096,-79.165,-176.126,8.652,148.597
C03277=1178.708,366.849,-79.131,-176.127,8.649,148.597
C03278=1178.711,366.601,-79.097,-176.129,8.646,148.597
C03279=1178.716,366.319,-79.057,-176.131,8.641,148.596
C03280=1178.721,366.038,-79.018,-176.133,8.638,148.596
C03281=1178.725,365.756,-78.979,-176.135,8.633,148.595
C03282=1178.730,365.475,-78.939,-176.137,8.630,148.595
C03283=1178.734,365.227,-78.905,-176.139,8.626,148.594
C03284=1178.738,364.979,-78.871,-176.141,8.622,148.594
C03285=1178.742,364.732,-78.837,-176.143,8.619,148.594
C03286=1178.746,364.484,-78.802,-176.145,8.616,148.593
C03287=1178.750,364.237,-78.768,-176.147,8.612,148.593
C03288=1178.754,363.989,-78.733,-176.148,8.608,148.592
C03289=1178.758,363.741,-78.700,-176.150,8.605,148.592
C03290=1178.762,363.493,-78.665,-176.152,8.601,148.592
C03291=1178.766,363.246,-78.631,-176.155,8.597,148.591
C03292=1178.770,362.998,-78.597,-176.157,8.593,148.591
C03293=1178.774,362.750,-78.562,-176.159,8.590,148.590
C03294=1178.778,362.503,-78.528,-176.160,8.586,148.590
C03295=1178.783,362.256,-78.494,-176.163,8.583,148.590
C03296=1178.786,362.008,-78.460,-176.164,8.579,148.589
C03297=1178.790,361.760,-78.426,-176.166,8.576,148.589
C03298=1178.794,361.512,-78.392,-176.169,8.572,148.589
C03299=1178.798,361.265,-78.358,-176.170,8.569,148.588
C03300=1178.802,361.018,-78.323,-176.173,8.565,148.588
C03301=1178.806,360.770,-78.289,-176.175,8.562,148.588
C03302=1178.810,360.522,-78.255,-176.176,8.558,148.587
C03303=1178.814,360.275,-78.221,-176.179,8.555,148.587
C03304=1178.818,360.027,-78.186,-176.180,8.551,148.587
C03305=1178.822,359.779,-78.153,-176.183,8.548,148.586
C03306=1178.826,359.532,-78.119,-176.185,8.543,148.586
C03307=1178.830,359.284,-78.085,-176.187,8.540,148.586
C03308=1178.834,359.036,-78.051,-176.189,8.536,148.585
C03309=1178.839,358.788,-78.017,-176.191,8.533,148.585
C03310=1178.842,358.541,-77.983,-176.193,8.530,148.585
C03311=1178.846,358.294,-77.949,-176.196,8.526,148.584
C03312=1178.851,358.045,-77.915,-176.198,8.523,148.584
C03313=1178.855,357.798,-77.881,-176.200,8.519,148.584
C03314=1178.858,357.550,-77.848,-176.202,8.516,148.583
C03315=1178.863,357.302,-77.813,-176.204,8.512,148.583
C03316=1178.867,357.055,-77.779,-176.207,8.508,148.583
C03317=1178.870,356.807,-77.746,-176.209,8.505,148.583
C03318=1178.875,356.560,-77.711,-176.211,8.501,148.582
C03319=1178.879,356.312,-77.678,-176.213,8.498,148.582
C03320=1178.883,356.065,-77.644,-176.215,8.495,148.582
C03321=1178.887,355.816,-77.610,-176.217,8.491,148.581
C03322=1178.891,355.569,-77.576,-176.219,8.488,148.581
C03323=1178.895,355.321,-77.543,-176.222,8.484,148.581
C03324=1178.899,355.074,-77.509,-176.224,8.480,148.580
C03325=1178.903,354.825,-77.475,-176.226,8.477,148.580
C03326=1178.907,354.578,-77.441,-176.228,8.473,148.580
C03327=1178.911,354.330,-77.408,-176.230,8.470,148.579
C03328=1178.915,354.083,-77.374,-176.233,8.466,148.579
C03329=1178.920,353.835,-77.341,-176.235,8.463,148.579
C03330=1178.923,353.587,-77.307,-176.237,8.460,148.579
C03331=1178.927,353.340,-77.273,-176.239,8.456,148.578
C03332=1178.931,353.092,-77.240,-176.241,8.453,148.578
C03333=1178.936,352.844,-77.206,-176.244,8.449,148.578
C03334=1178.940,352.597,-77.172,-176.246,8.445,148.578
C03335=1178.943,352.348,-77.139,-176.249,8.442,148.577
C03336=1178.948,352.101,-77.106,-176.250,8.438,148.577
C03337=1178.951,351.854,-77.072,-176.253,8.435,148.577
C03338=1178.956,351.606,-77.039,-176.255,8.432,148.577
C03339=1178.960,351.358,-77.005,-176.257,8.429,148.576
C03340=1178.964,351.111,-76.971,-176.259,8.425,148.576
C03341=1178.968,350.863,-76.938,-176.262,8.422,148.576
C03342=1178.972,350.615,-76.904,-176.264,8.418,148.575
C03343=1178.976,350.367,-76.871,-176.266,8.414,148.575
C03344=1178.980,350.119,-76.838,-176.269,8.411,148.575
C03345=1178.984,349.872,-76.804,-176.271,8.408,148.575
C03346=1178.988,349.624,-76.771,-176.273,8.404,148.575
C03347=1178.992,349.377,-76.738,-176.275,8.401,148.574
C03348=1178.997,349.128,-76.704,-176.278,8.398,148.574
C03349=1179.001,348.881,-76.671,-176.280,8.394,148.574
C03350=1179.005,348.632,-76.638,-176.282,8.391,148.574
C03351=1179.009,348.385,-76.604,-176.284,8.387,148.573
C03352=1179.013,348.137,-76.570,-176.286,8.384,148.573
C03353=1179.017,347.890,-76.537,-176.289,8.381,148.573
C03354=1179.021,347.642,-76.504,-176.291,8.377,148.573
C03355=1179.025,347.394,-76.471,-176.294,8.373,148.572
C03356=1179.029,347.147,-76.438,-176.296,8.370,148.572
C03357=1179.033,346.899,-76.405,-176.298,8.367,148.572
C03358=1179.038,346.651,-76.372,-176.300,8.363,148.572
C03359=1179.042,346.403,-76.338,-176.303,8.360,148.571
C03360=1179.046,346.156,-76.305,-176.305,8.357,148.571
C03361=1179.050,345.908,-76.272,-176.307,8.353,148.571
C03362=1179.054,345.660,-76.239,-176.310,8.350,148.571
C03363=1179.058,345.412,-76.206,-176.312,8.347,148.571
C03364=1179.062,345.165,-76.173,-176.314,8.344,148.570
C03365=1179.067,344.917,-76.139,-176.316,8.340,148.570
C03366=1179.071,344.669,-76.106,-176.319,8.337,148.570
C03367=1179.074,344.422,-76.074,-176.321,8.334,148.570
C03368=1179.078,344.174,-76.041,-176.323,8.330,148.570
C03369=1179.083,343.926,-76.008,-176.326,8.326,148.569
C03370=1179.087,343.678,-75.975,-176.328,8.323,148.569
C03371=1179.091,343.430,-75.942,-176.330,8.320,148.569
C03372=1179.095,343.183,-75.909,-176.333,8.316,148.569
C03373=1179.099,342.935,-75.876,-176.335,8.313,148.569
C03374=1179.103,342.687,-75.842,-176.338,8.310,148.568
C03375=1179.108,342.439,-75.810,-176.340,8.307,148.568
C03376=1179.111,342.191,-75.777,-176.342,8.303,148.568
C03377=1179.115,341.944,-75.744,-176.345,8.300,148.568
C03378=1179.120,341.696,-75.711,-176.347,8.297,148.568
C03379=1179.124,341.448,-75.679,-176.349,8.293,148.567
C03380=1179.128,341.200,-75.645,-176.351,8.290,148.567
C03381=1179.132,340.952,-75.612,-176.354,8.287,148.567
C03382=1179.136,340.705,-75.580,-176.356,8.284,148.567
C03383=1179.141,340.425,-75.543,-176.359,8.280,148.567
C03384=1179.145,340.146,-75.506,-176.361,8.276,148.566
C03385=1179.150,339.867,-75.469,-176.364,8.272,148.566
C03386=1179.155,339.589,-75.433,-176.367,8.269,148.566
C03387=1179.159,339.341,-75.399,-176.369,8.266,148.566
C03388=1179.163,339.092,-75.367,-176.372,8.262,148.566
C03389=1179.167,338.845,-75.334,-176.374,8.258,148.565
C03390=1179.171,338.597,-75.302,-176.377,8.255,148.565
C03391=1179.175,338.349,-75.269,-176.379,8.252,148.565
C03392=1179.179,338.101,-75.236,-176.381,8.248,148.565
C03393=1179.183,337.853,-75.204,-176.384,8.245,148.565
C03394=1179.187,337.605,-75.171,-176.386,8.242,148.565
C03395=1179.192,337.357,-75.138,-176.388,8.239,148.564
C03396=1179.196,337.110,-75.106,-176.391,8.236,148.564
C03397=1179.200,336.862,-75.074,-176.393,8.232,148.564
C03398=1179.204,336.614,-75.040,-176.396,8.229,148.564
C03399=1179.208,336.366,-75.009,-176.398,8.226,148.564
C03400=1179.212,336.119,-74.975,-176.400,8.223,148.564
C03401=1179.217,335.870,-74.943,-176.402,8.219,148.563
C03402=1179.220,335.623,-74.910,-176.405,8.216,148.563
C03403=1179.225,335.375,-74.878,-176.407,8.213,148.563
C03404=1179.229,335.127,-74.847,-176.410,8.210,148.563
C03405=1179.233,334.879,-74.813,-176.412,8.206,148.563
C03406=1179.237,334.631,-74.781,-176.415,8.203,148.563
C03407=1179.241,334.384,-74.748,-176.417,8.200,148.562
C03408=1179.245,334.135,-74.716,-176.419,8.197,148.562
C03409=1179.249,333.888,-74.684,-176.422,8.194,148.562
C03410=1179.254,333.640,-74.651,-176.424,8.190,148.562
C03411=1179.257,333.392,-74.619,-176.426,8.187,148.562
C03412=1179.262,333.144,-74.587,-176.429,8.184,148.562
C03413=1179.266,332.895,-74.555,-176.431,8.181,148.562
C03414=1179.270,332.649,-74.522,-176.434,8.178,148.561
C03415=1179.275,332.400,-74.490,-176.436,8.174,148.561
C03416=1179.278,332.152,-74.458,-176.439,8.171,148.561
C03417=1179.282,331.905,-74.425,-176.441,8.168,148.561
C03418=1179.287,331.657,-74.394,-176.443,8.165,148.561
C03419=1179.291,331.409,-74.361,-176.446,8.162,148.561
C03420=1179.295,331.161,-74.329,-176.448,8.158,148.561
C03421=1179.299,330.913,-74.297,-176.451,8.155,148.561
C03422=1179.303,330.666,-74.265,-176.453,8.152,148.560
C03423=1179.307,330.418,-74.233,-176.455,8.149,148.560
C03424=1179.311,330.169,-74.200,-176.458,8.146,148.560
C03425=1179.315,329.921,-74.168,-176.460,8.142,148.560
C03426=1179.320,329.674,-74.136,-176.463,8.139,148.560
C03427=1179.324,329.426,-74.105,-176.465,8.136,148.560
C03428=1179.328,329.178,-74.073,-176.468,8.133,148.560
C03429=1179.333,328.930,-74.041,-176.470,8.129,148.559
C03430=1179.336,328.682,-74.009,-176.473,8.126,148.559
C03431=1179.341,328.434,-73.976,-176.475,8.123,148.559
C03432=1179.345,328.186,-73.945,-176.478,8.120,148.559
C03433=1179.349,327.939,-73.912,-176.480,8.117,148.559
C03434=1179.353,327.690,-73.880,-176.483,8.114,148.559
C03435=1179.357,327.442,-73.848,-176.485,8.111,148.559
C03436=1179.361,327.195,-73.817,-176.487,8.107,148.559
C03437=1179.366,326.946,-73.785,-176.490,8.104,148.559
C03438=1179.369,326.698,-73.753,-176.492,8.101,148.558
C03439=1179.374,326.451,-73.721,-176.495,8.098,148.558
C03440=1179.378,326.202,-73.689,-176.497,8.095,148.558
C03441=1179.383,325.955,-73.658,-176.500,8.092,148.558
C03442=1179.386,325.707,-73.626,-176.502,8.088,148.558
C03443=1179.391,325.459,-73.593,-176.504,8.085,148.558
C03444=1179.395,325.211,-73.562,-176.507,8.082,148.558
C03445=1179.399,324.963,-73.530,-176.509,8.079,148.558
C03446=1179.402,324.715,-73.498,-176.512,8.076,148.558
C03447=1179.408,324.467,-73.467,-176.514,8.072,148.557
C03448=1179.411,324.219,-73.435,-176.517,8.069,148.557
C03449=1179.415,323.971,-73.403,-176.519,8.066,148.557
C03450=1179.419,323.724,-73.372,-176.522,8.063,148.557
C03451=1179.423,323.476,-73.340,-176.524,8.060,148.557
C03452=1179.428,323.228,-73.308,-176.527,8.057,148.557
C03453=1179.432,322.979,-73.277,-176.529,8.053,148.557
C03454=1179.436,322.731,-73.245,-176.532,8.050,148.557
C03455=1179.440,322.484,-73.213,-176.534,8.047,148.557
C03456=1179.444,322.235,-73.182,-176.537,8.044,148.557
C03457=1179.449,321.988,-73.151,-176.539,8.041,148.556
C03458=1179.453,321.740,-73.118,-176.542,8.038,148.556
C03459=1179.457,321.492,-73.087,-176.544,8.035,148.556
C03460=1179.461,321.244,-73.056,-176.547,8.032,148.556
C03461=1179.466,320.996,-73.024,-176.549,8.028,148.556
C03462=1179.469,320.748,-72.992,-176.552,8.025,148.556
C03463=1179.473,320.499,-72.961,-176.554,8.022,148.556
C03464=1179.478,320.252,-72.930,-176.557,8.019,148.556
C03465=1179.482,320.003,-72.898,-176.559,8.016,148.556
C03466=1179.486,319.756,-72.867,-176.561,8.013,148.556
C03467=1179.490,319.508,-72.835,-176.564,8.010,148.555
C03468=1179.495,319.260,-72.804,-176.566,8.007,148.555
C03469=1179.499,319.012,-72.772,-176.569,8.004,148.555
C03470=1179.503,318.764,-72.741,-176.571,8.001,148.555
C03471=1179.507,318.516,-72.709,-176.574,7.998,148.555
C03472=1179.512,318.268,-72.679,-176.576,7.995,148.555
C03473=1179.515,318.020,-72.647,-176.579,7.992,148.555
C03474=1179.520,317.772,-72.616,-176.581,7.988,148.555
C03475=1179.524,317.524,-72.584,-176.584,7.985,148.555
C03476=1179.528,317.276,-72.553,-176.587,7.982,148.555
C03477=1179.532,317.028,-72.522,-176.589,7.979,148.555
C03478=1179.537,316.780,-72.491,-176.592,7.976,148.555
C03479=1179.541,316.531,-72.460,-176.594,7.973,148.555
C03480=1179.545,316.284,-72.428,-176.597,7.970,148.555
C03481=1179.550,316.036,-72.397,-176.599,7.967,148.555
C03482=1179.553,315.788,-72.366,-176.602,7.963,148.554
C03483=1179.558,315.540,-72.335,-176.604,7.960,148.554
C03484=1179.561,315.292,-72.304,-176.607,7.957,148.554
C03485=1179.565,315.044,-72.273,-176.609,7.955,148.554
C03486=1179.569,314.796,-72.242,-176.612,7.952,148.554
C03487=1179.575,314.519,-72.207,-176.614,7.948,148.554
C03488=1179.579,314.242,-72.173,-176.617,7.945,148.554
C03489=1179.584,313.966,-72.138,-176.620,7.941,148.554
C03490=1179.589,313.689,-72.103,-176.623,7.938,148.554
C03491=1179.593,313.441,-72.072,-176.625,7.935,148.554
C03492=1179.597,313.192,-72.041,-176.628,7.932,148.554
C03493=1179.602,312.945,-72.010,-176.630,7.928,148.554
C03494=1179.606,312.697,-71.979,-176.633,7.925,148.554
C03495=1179.609,312.449,-71.948,-176.636,7.922,148.554
C03496=1179.614,312.201,-71.917,-176.638,7.919,148.553
C03497=1179.618,311.952,-71.886,-176.640,7.917,148.553
C03498=1179.622,311.705,-71.855,-176.643,7.914,148.553
C03499=1179.627,311.457,-71.824,-176.645,7.911,148.553
C03500=1179.630,311.208,-71.794,-176.648,7.908,148.553
C03501=1179.635,310.961,-71.763,-176.650,7.904,148.553
C03502=1179.639,310.713,-71.732,-176.653,7.901,148.553
C03503=1179.643,310.464,-71.701,-176.656,7.898,148.553
C03504=1179.648,310.216,-71.670,-176.658,7.895,148.553
C03505=1179.652,309.968,-71.640,-176.661,7.892,148.553
C03506=1179.656,309.720,-71.609,-176.663,7.889,148.553
C03507=1179.661,309.472,-71.578,-176.666,7.886,148.553
C03508=1179.665,309.224,-71.547,-176.668,7.883,148.553
C03509=1179.669,308.976,-71.517,-176.671,7.880,148.553
C03510=1179.673,308.727,-71.486,-176.673,7.877,148.553
C03511=1179.678,308.479,-71.455,-176.675,7.874,148.553
C03512=1179.682,308.232,-71.425,-176.678,7.871,148.553
C03513=1179.686,307.983,-71.394,-176.681,7.868,148.553
C03514=1179.690,307.735,-71.363,-176.683,7.865,148.553
C03515=1179.694,307.488,-71.333,-176.686,7.862,148.553
C03516=1179.699,307.240,-71.302,-176.689,7.859,148.553
C03517=1179.703,306.991,-71.271,-176.691,7.856,148.552
C03518=1179.707,306.743,-71.241,-176.694,7.853,148.552
C03519=1179.711,306.495,-71.210,-176.696,7.850,148.552
C03520=1179.716,306.247,-71.179,-176.699,7.847,148.552
C03521=1179.719,305.999,-71.149,-176.701,7.844,148.552
C03522=1179.724,305.750,-71.119,-176.704,7.841,148.552
C03523=1179.729,305.502,-71.088,-176.706,7.838,148.552
C03524=1179.732,305.255,-71.058,-176.709,7.835,148.552
C03525=1179.737,305.007,-71.027,-176.711,7.832,148.552
C03526=1179.740,304.759,-70.997,-176.714,7.829,148.552
C03527=1179.745,304.510,-70.967,-176.717,7.826,148.552
C03528=1179.750,304.262,-70.936,-176.719,7.823,148.552
C03529=1179.754,304.014,-70.906,-176.721,7.820,148.552
C03530=1179.758,303.766,-70.875,-176.724,7.817,148.552
C03531=1179.762,303.517,-70.845,-176.727,7.814,148.552
C03532=1179.767,303.269,-70.814,-176.729,7.811,148.552
C03533=1179.770,303.022,-70.784,-176.732,7.808,148.552
C03534=1179.775,302.773,-70.754,-176.734,7.805,148.552
C03535=1179.779,302.526,-70.724,-176.737,7.802,148.552
C03536=1179.784,302.278,-70.693,-176.740,7.799,148.552
C03537=1179.787,302.029,-70.663,-176.742,7.796,148.552
C03538=1179.792,301.781,-70.633,-176.744,7.794,148.552
C03539=1179.796,301.533,-70.602,-176.747,7.791,148.552
C03540=1179.801,301.284,-70.572,-176.750,7.788,148.552
C03541=1179.805,301.037,-70.542,-176.752,7.784,148.552
C03542=1179.810,300.788,-70.512,-176.755,7.781,148.552
C03543=1179.814,300.541,-70.482,-176.757,7.778,148.552
C03544=1179.817,300.292,-70.451,-176.760,7.775,148.552
C03545=1179.822,300.044,-70.421,-176.763,7.772,148.552
C03546=1179.826,299.796,-70.391,-176.764,7.770,148.552
C03547=1179.831,299.547,-70.361,-176.767,7.767,148.552
C03548=1179.834,299.300,-70.331,-176.770,7.764,148.552
C03549=1179.839,299.051,-70.301,-176.773,7.761,148.552
C03550=1179.843,298.804,-70.271,-176.775,7.758,148.552
C03551=1179.847,298.555,-70.241,-176.778,7.755,148.552
C03552=1179.852,298.307,-70.211,-176.780,7.752,148.552
C03553=1179.856,298.059,-70.181,-176.782,7.750,148.552
C03554=1179.860,297.811,-70.152,-176.785,7.747,148.552
C03555=1179.864,297.562,-70.121,-176.788,7.744,148.552
C03556=1179.869,297.314,-70.091,-176.790,7.740,148.552
C03557=1179.872,297.066,-70.061,-176.793,7.737,148.552
C03558=1179.877,296.818,-70.031,-176.796,7.734,148.552
C03559=1179.882,296.569,-70.001,-176.798,7.731,148.552
C03560=1179.885,296.322,-69.971,-176.801,7.729,148.552
C03561=1179.890,296.073,-69.942,-176.803,7.726,148.552
C03562=1179.894,295.825,-69.912,-176.806,7.723,148.552
C03563=1179.898,295.577,-69.882,-176.808,7.720,148.552
C03564=1179.903,295.329,-69.852,-176.811,7.717,148.552
C03565=1179.907,295.081,-69.823,-176.814,7.714,148.552
C03566=1179.911,294.833,-69.792,-176.816,7.711,148.552
C03567=1179.916,294.585,-69.762,-176.819,7.709,148.552
C03568=1179.920,294.336,-69.733,-176.821,7.705,148.552
C03569=1179.924,294.088,-69.704,-176.824,7.702,148.552
C03570=1179.929,293.840,-69.673,-176.826,7.699,148.552
C03571=1179.933,293.592,-69.643,-176.829,7.696,148.552
C03572=1179.937,293.343,-69.614,-176.832,7.693,148.552
C03573=1179.941,293.095,-69.584,-176.834,7.691,148.552
C03574=1179.945,292.847,-69.555,-176.837,7.688,148.552
C03575=1179.949,292.599,-69.526,-176.839,7.685,148.552
C03576=1179.954,292.351,-69.495,-176.842,7.682,148.552
C03577=1179.958,292.102,-69.465,-176.844,7.679,148.552
C03578=1179.962,291.854,-69.436,-176.847,7.676,148.552
C03579=1179.967,291.606,-69.406,-176.849,7.674,148.552
C03580=1179.971,291.358,-69.377,-176.852,7.671,148.552
C03581=1179.975,291.109,-69.347,-176.855,7.668,148.552
C03582=1179.979,290.861,-69.318,-176.857,7.665,148.552
C03583=1179.984,290.614,-69.289,-176.860,7.662,148.552
C03584=1179.989,290.365,-69.259,-176.862,7.659,148.552
C03585=1179.993,290.117,-69.229,-176.865,7.656,148.552
C03586=1179.997,289.868,-69.200,-176.867,7.653,148.552
C03587=1180.001,289.620,-69.171,-176.870,7.650,148.552
C03588=1180.006,289.372,-69.141,-176.873,7.647,148.552
C03589=1180.010,289.124,-69.112,-176.876,7.644,148.552
C03590=1180.014,288.875,-69.082,-176.878,7.642,148.552
C03591=1180.019,288.601,-69.049,-176.881,7.638,148.552
C03592=1180.023,288.326,-69.017,-176.884,7.635,148.552
C03593=1180.028,288.051,-68.985,-176.886,7.633,148.552
C03594=1180.033,287.777,-68.952,-176.889,7.630,148.552
C03595=1180.037,287.529,-68.923,-176.892,7.627,148.552
C03596=1180.041,287.281,-68.893,-176.895,7.624,148.552
C03597=1180.046,287.032,-68.865,-176.897,7.621,148.552
C03598=1180.050,286.783,-68.835,-176.899,7.618,148.552
C03599=1180.055,286.536,-68.806,-176.902,7.615,148.552
C03600=1180.059,286.288,-68.777,-176.904,7.612,148.552
C03601=1180.063,286.039,-68.747,-176.907,7.609,148.552
C03602=1180.067,285.791,-68.718,-176.910,7.606,148.552
C03603=1180.072,285.542,-68.689,-176.912,7.604,148.552
C03604=1180.076,285.295,-68.660,-176.915,7.601,148.552
C03605=1180.081,285.046,-68.630,-176.918,7.598,148.552
C03606=1180.085,284.798,-68.601,-176.920,7.595,148.552
C03607=1180.089,284.549,-68.572,-176.923,7.592,148.552
C03608=1180.093,284.301,-68.543,-176.925,7.590,148.552
C03609=1180.097,284.054,-68.514,-176.928,7.587,148.552
C03610=1180.102,283.805,-68.486,-176.931,7.584,148.552
C03611=1180.106,283.557,-68.456,-176.933,7.581,148.552
C03612=1180.110,283.308,-68.427,-176.936,7.579,148.553
C03613=1180.115,283.059,-68.398,-176.938,7.576,148.553
C03614=1180.120,282.812,-68.369,-176.941,7.573,148.553
C03615=1180.124,282.564,-68.339,-176.944,7.570,148.553
C03616=1180.128,282.315,-68.311,-176.946,7.567,148.553
C03617=1180.132,282.067,-68.282,-176.948,7.564,148.553
C03618=1180.137,281.819,-68.253,-176.951,7.561,148.553
C03619=1180.141,281.570,-68.224,-176.954,7.558,148.553
C03620=1180.145,281.322,-68.194,-176.956,7.555,148.553
C03621=1180.150,281.074,-68.167,-176.959,7.553,148.553
C03622=1180.154,280.826,-68.137,-176.961,7.550,148.553
C03623=1180.158,280.577,-68.109,-176.964,7.547,148.553
C03624=1180.162,280.329,-68.079,-176.967,7.544,148.553
C03625=1180.167,280.081,-68.051,-176.969,7.542,148.553
C03626=1180.171,279.833,-68.022,-176.972,7.539,148.553
C03627=1180.175,279.584,-67.993,-176.974,7.536,148.553
C03628=1180.180,279.335,-67.964,-176.977,7.533,148.553
C03629=1180.184,279.087,-67.936,-176.980,7.530,148.553
C03630=1180.188,278.839,-67.906,-176.982,7.528,148.553
C03631=1180.193,278.590,-67.878,-176.985,7.525,148.553
C03632=1180.197,278.342,-67.850,-176.987,7.522,148.553
C03633=1180.201,278.094,-67.820,-176.990,7.519,148.553
C03634=1180.206,277.845,-67.792,-176.992,7.517,148.553
C03635=1180.210,277.598,-67.763,-176.995,7.514,148.553
C03636=1180.214,277.349,-67.734,-176.998,7.511,148.553
C03637=1180.219,277.100,-67.706,-177.000,7.509,148.554
C03638=1180.223,276.853,-67.677,-177.003,7.506,148.554
C03639=1180.227,276.604,-67.649,-177.005,7.503,148.554
C03640=1180.231,276.356,-67.620,-177.008,7.500,148.554
C03641=1180.236,276.108,-67.591,-177.011,7.498,148.554
C03642=1180.240,275.859,-67.563,-177.013,7.495,148.554
C03643=1180.245,275.611,-67.535,-177.016,7.492,148.554
C03644=1180.249,275.362,-67.506,-177.019,7.489,148.554
C03645=1180.252,275.114,-67.477,-177.021,7.487,148.554
C03646=1180.258,274.866,-67.449,-177.024,7.484,148.554
C03647=1180.262,274.617,-67.420,-177.027,7.481,148.554
C03648=1180.266,274.369,-67.392,-177.029,7.478,148.554
C03649=1180.271,274.121,-67.363,-177.031,7.476,148.554
C03650=1180.274,273.873,-67.335,-177.034,7.473,148.554
C03651=1180.279,273.624,-67.306,-177.037,7.470,148.554
C03652=1180.283,273.376,-67.278,-177.039,7.468,148.555
C03653=1180.288,273.128,-67.250,-177.042,7.465,148.555
C03654=1180.292,272.879,-67.222,-177.045,7.462,148.555
C03655=1180.297,272.631,-67.193,-177.047,7.459,148.555
C03656=1180.301,272.383,-67.164,-177.049,7.457,148.555
C03657=1180.305,272.134,-67.136,-177.052,7.454,148.555
